(* CODESYS project tc3_bacnetrev14.library
   Company: Beckhoff Automation GmbH
   DefaultNamespace: Tc3_BACnetRev14
   Version: 4.0.11.0
   Placeholder: Tc3_BACnetRev14
   Author: Beckhoff Automation GmbH
   Description: The PLC library is a collection of function blocks for programming a BACnet controller. For each BACnet object function blocks are available that are read and written via the selected properties. In general a distinction is made between function blocks for server and client objects. Function blocks for client objects have the prefix "Remote", since they enable access to remote BACnet objects on other devices. The BACnet object function blocks ascertain whether process data are valid and the BACnet controller is ready for operation.
   Title: Tc3_BACnetRev14

Project tree, tasks and I/O mapping:
  libraries: Tc2_Standard, * (Beckhoff Automation GmbH); Tc2_System, * (Beckhoff Automation GmbH); Tc2_Utilities, * (Beckhoff Automation GmbH); Tc3_BA2_Common, * (Beckhoff Automation GmbH); Tc3_Module, * (Beckhoff Automation GmbH)
  DUTs/
    Enumerations/
      [Internal]/
        data type E_BACnet_CommMode
        data type E_BACnet_MultistateVal
        data type E_BACnet_PlcAction
      Properties/
        Calendar/
          data type E_BACnet_CalendarEntryChoice
          data type E_BACnet_CalendarEntryType
        DateTime/
          data type E_BACnet_DaysOfWeekBits
          data type E_BACnet_TimeStampChoice
        Error/
          data type E_BACnet_ErrorClass
          data type E_BACnet_ErrorCode
          data type E_BACnet_ErrorType
        Event/
          data type E_BACnet_EventState
          data type E_BACnet_EventTransitionBits
          data type E_BACnet_EventType
        LogBuffer/
          data type E_BACnet_LogRecordChoice
        Recipient/
          data type E_BACnet_AddressChoice
          data type E_BACnet_RecipientChoice
        Scheduler/
          data type E_BACnet_EnumerationValueChoice
          data type E_BACnet_SchedBType
          data type E_BACnet_SpecialEventChoice
          data type E_BACnet_ValueChoice
        data type E_BACnet_AbortReason
        data type E_BACnet_AdapterStatus
        data type E_BACnet_BinaryPV
        data type E_BACnet_DataTypes
        data type E_BACnet_DeviceStatus
        data type E_BACnet_FileAccessMethod
        data type E_BACnet_LifeSafetyMode
        data type E_BACnet_LifeSafetyOperation
        data type E_BACnet_LimitEnableBits
        data type E_BACnet_LoopMode
        data type E_BACnet_NodeType
        data type E_BACnet_NotifyType
        data type E_BACnet_ObjectSupportedBits
        data type E_BACnet_PersistentDataState
        data type E_BACnet_Priority
        data type E_BACnet_ProgramError
        data type E_BACnet_ProgramRequest
        data type E_BACnet_ProgramState
        data type E_BACnet_RejectReason
        data type E_BACnet_Reliability
        data type E_BACnet_Segmentation
        data type E_BACnet_ServicesSupportedBits
        data type E_BACnet_SilencedState
        data type E_BACnet_StatusFlags
        data type E_BACnet_StringEncodingTypes
      Remote/
        data type E_BACnetRM_ClientState
        data type E_BACnetRM_Error
        data type E_BACnetRM_RequestType
      data type E_BACnet_Error
    Interfaces/
      Remote/
        [Base]/
          interface I_BACnetRM_Object
        [Internal]/
          interface I_BACnetRM_BaseObject: OnCOV, OnReqError, Error, ObjectID, ObjectInstance, ObjectType, Ready
          interface I_BACnetRM_ObjectOwner: OnBACnetRMObjectCOV, OnBACnetRMObjectStateChanged, LogMsg
        interface I_BACnetRM_Req: Send, GetRequestType, IsReady
      Server/
        [Base]/
          interface I_BACnet_Object: Parent, Description, ObjectName
        [Internal]/
          interface I_BACnet_BaseObject: Error, ObjectID, ObjectInstance, ObjectType, Ready, ReadProperty, SyncPropertyCOV, WriteProperty
          interface I_BACnet_ObjectOwner: OnBACnetObjectStateChanged, LogMsg, SymbolPath
        Misc/
          interface I_BACnet_Cal
          interface I_BACnet_View
    Types/
      [ADS]/
        data type ST_BACnet_AdsConnection
        data type ST_BACnet_GlobalAdsBuffer
      [Internal]/
        ObjectList/
          data type ST_ObjectListEntry
      Diagnose/
        data type ST_BACnet_ConfirmedServiceDiag
        data type ST_BACnet_DiagEthStatistics
        data type ST_BACnet_Diagnosis
        data type ST_BACnet_DiagnosisTiming
        data type ST_BACnet_FrameStatistics
        data type ST_BACnet_Info
        data type ST_BACnet_ServerStatistics
        data type ST_BACnet_TcIoEthStatistic
        data type ST_BACnet_TcIoEthTxRxErrorCount
        data type ST_BACnet_UnConfirmedServiceDiag
      Properties/
        [ADS]/
          Calendar/
            data type ST_BACnet_CalendarEntry
            data type ST_BACnet_CalendarEntryDate
            data type ST_BACnet_CalendarEntryDateRange
            data type ST_BACnet_CalendarEntryWeekNDay
            data type T_BACnet_CalendarEntryTypeFilter
          DateTime/
            data type ST_BACnet_TimeStampDateTime
            data type ST_BACnet_TimeValue
            data type ST_BACnet_TimeValueBool
            data type ST_BACnet_TimeValueList
            data type ST_BACnet_TimeValueReal
          LogBuffer/
            data type ST_BACnet_LogBufferEntryReal
            data type ST_BACnet_LogBufferReal
          LogRecord/
            data type ST_BACnet_LogDatum
            data type ST_BACnet_LogDatumList
            data type ST_BACnet_LogRecord
            data type ST_BACnet_LogRecordList
          Schedule/
            data type ST_BACnet_DailySchedule
            data type ST_BACnet_ExceptionScheduleBool
            data type ST_BACnet_ExceptionScheduleCalDate
            data type ST_BACnet_ExceptionScheduleCalRef
            data type ST_BACnet_ExceptionScheduleCalWnD
            data type ST_BACnet_ExceptionScheduleEntryBool
            data type ST_BACnet_ExceptionScheduleEntryReal
            data type ST_BACnet_ExceptionScheduleReal
            data type ST_BACnet_Value
            data type ST_BACnet_ValueList
            data type ST_BACnet_WeeklyScheduleBool
            data type ST_BACnet_WeeklyScheduleReal
          ValidFields/
            data type ST_BACnet_ValidFields_DeviceObjectPropertyReference
          data type ST_BACnet_CharacterStringExt
          data type ST_BACnet_CharacterStringExtListEntry
          data type ST_BACnet_DeviceObjectPropertyReference
          data type ST_BACnet_DeviceObjectReference
          data type ST_BACnet_LimitEnable
          data type ST_BACnet_ObjectIdentifierList
        Calendar/
          data type T_BACnet_CalendarDateList
        Event/
          data type ST_BACnet_Event
          data type ST_BACnet_EventMessageTexts
          data type ST_BACnet_EventMessageTextStrings
          data type ST_BACnet_Events
          data type ST_BACnet_EventTimeStamps
        Recipient/
          data type ST_BACnet_Address
          data type ST_BACnet_Destination
          data type ST_BACnet_Recipient
          data type ST_BACnet_RecipientEntry
          data type ST_BACnet_ValidDays
        References/
          data type ST_BACnet_ObjectPropertyReference
        Scheduler/
          data type ST_BACnet_EnumerationValueType
          data type ST_BACnet_SchedCalendar
          data type ST_BACnet_SchedException
          data type ST_BACnet_SpecialEvent
          data type ST_BACnet_SpecialEventList
          data type T_BACnet_SchedCalendar
          data type T_BACnet_SchedExceptionEntryList
          data type T_BACnet_SchedExceptionList
          data type T_BACnet_SchedWeek
        TLog/
          data type T_BACnet_TLogBuffer
        data type ST_BACnet_EventTransitionBits
        data type ST_BACnet_ServicesSupportedBits
        data type T_BACnet_ObjectIdentifier
        data type T_BACnet_StateText
      Remote/
        [Internal]/
          data type ST_BACnetRM_CmdRealValue
          data type ST_BACnetRM_FifoEntry
          data type ST_BACnetRM_LastWriteValue
          data type ST_BACnetRM_PropertyValueList
          data type ST_BACnetRM_ReadEntry
          data type ST_BACnetRM_ReqPtr
          data type ST_BACnetRM_RpmListEntry
          data type ST_BACnetRM_ScanParameter
          data type ST_BACnetRM_WriteEntry
        data type ST_BACnetRM_ScanResult
  GVLs/
    global variables BACnet_Globals
    global variables BACnet_Param
  POUs/
    Helper/
      [internal]/
        Calendar/
          function F_BACnet_CopyDateListEntry [ST]
        Remote/
          function F_BACnetRM_IsErrorSet [ST]
        String/
          function F_BACnet_ChrStrExtLen [ST]
          function F_BACnet_DecodeUCS2 [ST]
          function F_BACnet_DecodeUCS4 [ST]
          function F_BACnet_DecodeUTF8 [ST]
          function F_BACnet_EncodeUTF8 [ST]
          function F_BACnet_GetUsedStateText [ST]
          function F_BACnet_GetUsedUDINT [ST]
          function F_BACnet_UCS2ToWin1252 [ST]
          function F_BACnet_Utf8ToWin1252 [ST]
          function F_BACnet_Win1252ToUCS2 [ST]
          function F_BACnet_Win1252ToUtf8 [ST]
        Validation-Functions/
          function F_BACnet_IsObjIdentifierValid [ST]
          function F_BACnet_IsPriorityValid [ST]
          function F_BACnet_IsSchedBTypeValid [ST]
        function F_BACnet_AlignedSize [ST]
        function F_BACnet_AnalogPV [ST]
        function F_BACnet_BitFieldBit [ST]
        function F_BACnet_ChangeBitFieldBit [ST]
        function F_BACnet_EndOf [ST]
        function F_BACnet_IsBitFieldBitSet [ST]
        function F_BACnet_IsBitFieldBitSetPtr [ST]
        function F_BACnet_NextListElem [ST]
        function F_BACnet_SetBitFieldBit [ST]
        function F_BACnet_SysTimeDiff [ST]
        function F_BACnet_UnSetBitFieldBit [ST]
      Flags/
        function F_BACnet_EventEnable [ST]
        function F_BACnet_EventTransitionFlags [ST]
        function F_BACnet_GetEventTransFlagsData [ST]
        function F_BACnet_GetLimitEnFlagsData [ST]
        function F_BACnet_GetStatusFlagsData [ST]
        function F_BACnet_LimitEnable [ST]
        function F_BACnet_LimitEnableFlags [ST]
        function F_BACnet_StatusFlags [ST]
      MultiState/
        function F_BACnet_EnMultiStatePV [ST]
        function F_BACnet_MultiStatePV [ST]
      NC/
        function F_BACnet_DeviceRecipient [ST]
        function F_BACnet_EthernetRecipient [ST]
        function F_BACnet_EthernetRecipientEx [ST]
      Real/
        function F_BACnet_EnRealPV [ST]
        function F_BACnet_IsFinite [ST]
        function F_BACnet_NAN [ST]
        function F_BACnet_RealEQ [ST]
        function F_BACnet_RealGE [ST]
        function F_BACnet_RealGT [ST]
        function F_BACnet_RealLE [ST]
        function F_BACnet_RealLT [ST]
        function F_BACnet_RealNothing [ST]
        function F_BACnet_RealNull [ST]
        function F_BACnet_RealPV [ST]
        function F_BACnet_RealToStr [ST]
      Scheduler/
        Calendar/
          function F_BACnet_SchedCalendar [ST]
        Exception/
          function F_BACnet_SchedEntry1xA [ST]
          function F_BACnet_SchedEntry1xB [ST]
          function F_BACnet_SchedEntry1xM [ST]
          function F_BACnet_SchedEntry3xA [ST]
          function F_BACnet_SchedEntry3xB [ST]
          function F_BACnet_SchedEntry3xM [ST]
          function F_BACnet_SchedEntry5xA [ST]
          function F_BACnet_SchedEntry5xB [ST]
          function F_BACnet_SchedEntry5xM [ST]
        Weekly/
          function F_BACnet_SchedWeekly1xA [ST]
          function F_BACnet_SchedWeekly1xB [ST]
          function F_BACnet_SchedWeekly1xM [ST]
          function F_BACnet_SchedWeekly3xA [ST]
          function F_BACnet_SchedWeekly3xB [ST]
          function F_BACnet_SchedWeekly3xM [ST]
          function F_BACnet_SchedWeekly5xA [ST]
          function F_BACnet_SchedWeekly5xB [ST]
          function F_BACnet_SchedWeekly5xM [ST]
      String/
        function F_BACnet_GetObjectIdString [ST]
        function block FB_BACnet_StringExtDecode [ST]
        function block FB_BACnet_StringExtEncode [ST]
      function F_BACnet_GetObjectListIndex [ST]
      function F_BACnet_GetObjId [ST]
      function F_BACnet_GetObjInstance [ST]
      function F_BACnet_GetObjType [ST]
      function block FB_BACnet_AccLimit [ST]
      function block FB_BACnet_AvgValue [ST]
      function block FB_BACnet_PidControl [ST]
      function block FB_BACnet_PT1 [ST]
    Local/
      Objects/
        [Base]/
          Basic/
            function block FB_BACnet_EventObject [ST]: OnObjectStateChanged, FB_init, AcknowledgePLC, AcknowledgeRm, IsReliable, AckedTransitions, EventState, StateFlags
            function block FB_BACnet_Object [ST]: OnBACnetObjectStateChanged, OnObjectStateChanged, ValidateReference, ConcatTitle, ValidateTitles, FB_init, LogMsg, Parent, SymbolPath, ReadPropertyExceptionSched, ReadPropertyReference, WritePropertyExceptionSched, WritePropertyReference, Description, ObjectName
          function block FB_BACnet_BaseAI [ST]: OnObjectStateChanged, FB_init
          function block FB_BACnet_BaseAO [ST]: OnObjectStateChanged, FB_init
          function block FB_BACnet_BaseBI [ST]: OnObjectStateChanged, FB_init
          function block FB_BACnet_BaseBO [ST]: OnObjectStateChanged, FB_init
          function block FB_BACnet_BaseMI [ST]: OnObjectStateChanged, FB_init, StateCount
          function block FB_BACnet_BaseMO [ST]: OnObjectStateChanged, FB_init, StateCount
          function block FB_BACnet_BaseSched [ST]: OnObjectStateChanged, FB_init, ReadContent, WriteContent
          function block FB_BACnet_BaseTLog [ST]: OnObjectStateChanged
        [Internal]/
          Property/
            Buffer/
              [Archiv]/
                function block FB_BACnet_WeeklyScheduleBuffer [ST]: FB_init, ResetValue
              Base/
                function block FB_BACnet_BaseArrayBuffer [ST]
                function block FB_BACnet_BaseListBuffer [ST]: ValidateInst
                function block FB_BACnet_BasePropertyBuffer [ST]: ReadValue, WriteValue, MemSet, MemSetBYTE, MemSetUDINT, MemSetUINT, MemSetULINT, ValidateInst, OnObjectStateChanged, ResetValue
              function block FB_BACnet_DateListBuffer [ST]: FB_init
              function block FB_BACnet_EventLogBuffer [ST]: ValidateInst, FB_init
              function block FB_BACnet_ExceptionScheduleBuffer [ST]: FB_init
              function block FB_BACnet_TLMBuffer [ST]: ValidateInst, FB_init, ResetValue
              function block FB_BACnet_TrendLogBuffer [ST]: ValidateInst, FB_init, ResetValue
          function block FB_BACnet_BaseObject [ST]: Close, Execute, View_RegisterChildObject, DeleteObject, Sched_ReadEntry, Sched_SetNextDay, Sched_SetNextTimeVal, Sched_WriteEntry, Trend_NextLogRecord, OnObjectStateChanged, OnPostOnlineChange, FB_exit, Acknowledge, Error, ObjectID, ObjectInstance, ObjectType, Ready, State, EnableProperty, SetPropertyCount, WriteProtectProperty, AddPropertyElement, AddPropertyElementPtr, RemoveArrayElements, RemoveListElements, SetNumberOfStates, ReadProperty, ReadPropertyAckedTransitions, ReadPropertyBool, ReadPropertyDateList, ReadPropertyEventEnable, ReadPropertyEventState, ReadPropertyEventTimeStamps, ReadPropertyExceptionSched, ReadPropertyLimitEnable, ReadPropertyLogBuffer, ReadPropertyNotifyType, ReadPropertyReal, ReadPropertyRecipientList, ReadPropertyReference, ReadPropertyStatusFlags, ReadPropertyString, ReadPropertyUDInt, ReadPropertyUnit, ReadPropertyWeeklySched, GetSyncHandleMode, AddListElement, ApplySyncHandler, EvaluatePropSync, RequestSyncHandlers, RequestSyncHandlersEx, SyncProperty, SyncPropertyCOV, SyncPropertyIdx, SyncPropertyList, SyncPropertyPvPrio, WriteProperty, WritePropertyBool, WritePropertyDateList, WritePropertyEventEnable, WritePropertyExceptionSched, WritePropertyLimitEnable, WritePropertyLogBuffer, WritePropertyNotifyType, WritePropertyNull, WritePropertyReal, WritePropertyRealPrio, WritePropertyRecipientList, WritePropertyReference, WritePropertyString, WritePropertyStringIdx, WritePropertyUDInt, WritePropertyUInt, WritePropertyUnit, WritePropertyValue, WritePropertyValueEx, WritePropertyWeeklySched
        5P/
          function block FB_BACnet_AO_IO5P [ST]: OnObjectStateChanged, ActivePrio, EnManualRm, ValManualRm
          function block FB_BACnet_AO_Raw5P [ST]: OnObjectStateChanged, ActivePrio, EnManualRm, ValManualRm
          function block FB_BACnet_AV_5P [ST]: OnObjectStateChanged, ActivePrio, EnManualRm, ValManualRm
          function block FB_BACnet_BO_IO5P [ST]: OnObjectStateChanged, ActivePrio, EnManualRm, ValManualRm
          function block FB_BACnet_BO_Raw5P [ST]: OnObjectStateChanged, ActivePrio, EnManualRm, ValManualRm
          function block FB_BACnet_BV_5P [ST]: OnObjectStateChanged, ActivePrio, EnManualRm, ValManualRm
          function block FB_BACnet_MO_IO5P [ST]: OnObjectStateChanged, ActivePrio, EnManualRm, ValManualRm
          function block FB_BACnet_MO_Raw5P [ST]: OnObjectStateChanged, ActivePrio, EnManualRm, ValManualRm
          function block FB_BACnet_MV_5P [ST]: OnObjectStateChanged, ActivePrio, EnManualRm, ValManualRm
        function block FB_BACnet_Acc [ST]: OnObjectStateChanged, FB_init
        function block FB_BACnet_AI [ST]: OnObjectStateChanged
        function block FB_BACnet_AI_IO [ST]: OnObjectStateChanged
        function block FB_BACnet_AI_Raw [ST]: OnObjectStateChanged
        function block FB_BACnet_AO_IO [ST]: OnObjectStateChanged
        function block FB_BACnet_AO_Raw [ST]: OnObjectStateChanged
        function block FB_BACnet_AV [ST]: OnObjectStateChanged, FB_init
        function block FB_BACnet_AV_Disp [ST]: OnObjectStateChanged, FB_init
        function block FB_BACnet_AV_Setp [ST]: OnObjectStateChanged, FB_init
        function block FB_BACnet_BI_IO [ST]: OnObjectStateChanged
        function block FB_BACnet_BI_Raw [ST]: OnObjectStateChanged
        function block FB_BACnet_BO_IO [ST]: OnObjectStateChanged
        function block FB_BACnet_BO_Raw [ST]: OnObjectStateChanged
        function block FB_BACnet_BV [ST]: OnObjectStateChanged, FB_init
        function block FB_BACnet_BV_Disp [ST]: OnObjectStateChanged, FB_init
        function block FB_BACnet_BV_Setp [ST]: OnObjectStateChanged, FB_init
        function block FB_BACnet_Cal [ST]: OnObjectStateChanged, FB_init, ReadContent, WriteContent
        function block FB_BACnet_Device [ST]: OnObjectStateChanged, FB_init, Location
        function block FB_BACnet_EventLog [ST]: OnObjectStateChanged, FB_init
        function block FB_BACnet_Loop [ST]: OnObjectStateChanged, FB_init, Mode, ProportionalBand
        function block FB_BACnet_MI_IO [ST]
        function block FB_BACnet_MI_Raw [ST]
        function block FB_BACnet_MO_IO [ST]: OnObjectStateChanged
        function block FB_BACnet_MO_Raw [ST]
        function block FB_BACnet_MV [ST]: OnObjectStateChanged, FB_init, StateCount
        function block FB_BACnet_MV_Disp [ST]: OnObjectStateChanged, FB_init, StateCount
        function block FB_BACnet_MV_Setp [ST]: OnObjectStateChanged, FB_init, StateCount
        function block FB_BACnet_NC [ST]: OnObjectStateChanged, FB_init
        function block FB_BACnet_PC [ST]: OnObjectStateChanged, FB_init
        function block FB_BACnet_Prog [ST]: OnObjectStateChanged, FB_init
        function block FB_BACnet_SchedA [ST]: OnObjectStateChanged, FB_init
        function block FB_BACnet_SchedB [ST]: OnObjectStateChanged, FB_init
        function block FB_BACnet_SchedM [ST]: OnObjectStateChanged, FB_init
        function block FB_BACnet_TLM [ST]: OnObjectStateChanged, FB_init
        function block FB_BACnet_TLog [ST]: OnObjectStateChanged, FB_init, DeviceObjectPropertyReference
        function block FB_BACnet_View [ST]: OnObjectStateChanged, FB_init
      function block FB_BACnet_Server [ST]: GetObject, RegisterObject, ObjectCount, ServerItf, BackupSTM, Reset, OnPostOnlineChange, FB_Exit, Error, IsValid, ReadPropertyUint
    Remote/
      Objects/
        Basic/
          [Base]/
            Basic/
              function block FB_BACnetRM_Object [ST]: OnBACnetRMObjectCOV, OnBACnetRMObjectStateChanged, FB_init, LogMsg
            function block FB_BACnetRM_BaseTLog [ST]: OnObjectStateChanged
            function block FB_BACnetRM_EventObject [ST]: OnObjectStateChanged, StateFlags
          [Internal]/
            function block FB_BACnetRM_BaseObject [ST]: OnCOV, OnReqError, OnObjectStateChanged, Error, ObjectID, ObjectInstance, ObjectType, Ready, SyncProperty, SyncPropertyPrio
          function block FB_BACnetRM_Acc [ST]: OnObjectStateChanged, FB_init
          function block FB_BACnetRM_AI [ST]: OnObjectStateChanged, FB_init
          function block FB_BACnetRM_AO [ST]: OnObjectStateChanged, FB_init
          function block FB_BACnetRM_AV [ST]: OnObjectStateChanged, FB_init
          function block FB_BACnetRM_AV_Disp [ST]: OnObjectStateChanged, FB_init
          function block FB_BACnetRM_AV_Setp [ST]: OnCOV, OnObjectStateChanged, FB_init
          function block FB_BACnetRM_BI [ST]: OnObjectStateChanged, FB_init
          function block FB_BACnetRM_BO [ST]: OnObjectStateChanged, FB_init
          function block FB_BACnetRM_BV [ST]: OnObjectStateChanged, FB_init
          function block FB_BACnetRM_BV_Disp [ST]: OnObjectStateChanged, FB_init
          function block FB_BACnetRM_BV_Setp [ST]: OnCOV, OnObjectStateChanged, FB_init
          function block FB_BACnetRM_Cal [ST]: OnObjectStateChanged, FB_init
          function block FB_BACnetRM_Device [ST]: OnObjectStateChanged, FB_init
          function block FB_BACnetRM_Loop [ST]: OnObjectStateChanged, FB_init
          function block FB_BACnetRM_MI [ST]: OnObjectStateChanged, FB_init
          function block FB_BACnetRM_MO [ST]: OnObjectStateChanged, FB_init
          function block FB_BACnetRM_MV [ST]: OnObjectStateChanged, FB_init
          function block FB_BACnetRM_MV_Disp [ST]: OnObjectStateChanged, FB_init
          function block FB_BACnetRM_MV_Setp [ST]: OnCOV, OnObjectStateChanged, FB_init
          function block FB_BACnetRM_NC [ST]: OnObjectStateChanged, FB_init
          function block FB_BACnetRM_PC [ST]: OnObjectStateChanged, FB_init
          function block FB_BACnetRM_Prog [ST]: OnObjectStateChanged, FB_init
          function block FB_BACnetRM_SchedA [ST]: OnObjectStateChanged, FB_init
          function block FB_BACnetRM_SchedB [ST]: OnObjectStateChanged, FB_init
          function block FB_BACnetRM_SchedM [ST]: OnObjectStateChanged, FB_init
          function block FB_BACnetRM_TLM [ST]: FB_init
          function block FB_BACnetRM_TLog [ST]: FB_init
        Convenience/
          function block FB_BACnetRM_CnvLoop [ST]: OnObjectStateChanged
      Requests/
        [Internal]/
          [Base]/
            function block FB_BACnetRM_BaseProperty [ST]: OnExecuteChange, Free, Busy, Error, IsValid, Ready, Request
            function block FB_BACnetRM_ReqBase [ST]: GetRequestType, IsReady, IsValid, Send
            function block FB_BACnetRM_ReqBasic [ST]: OnSendPropertyDataRequest, InitTimer, TcAddRef, TcQueryInterface, TcRelease, OnError, CopyRemoteData, ProcessResult, Send, StartTimer, GetRequestType, IsReady
          function block FB_BACnetRM_ReqAckAlarm [ST]: OnSendPropertyDataRequest, Send, TcAddRef, TcQueryInterface, TcRelease, UpdateTimeStamp, GetRequestType, IsReady
          function block FB_BACnetRM_ReqCov [ST]: AddCovSlave, Send, ProcessResult, StartTimer, FB_Exit, GetRequestType, IsReady, Master, SendSubscription
          function block FB_BACnetRM_ReqFifo [ST]: AddFifoReq, ProcessReadFifo, ProcessWriteFifo, FB_Exit, IsValid
          function block FB_BACnetRM_ReqListAdd [ST]: Send, ProcessResult, GetRequestType, IsReady
          function block FB_BACnetRM_ReqListRem [ST]: Send, ProcessResult, GetRequestType
          function block FB_BACnetRM_ReqRead [ST]: Send, OnError, ProcessResult, GetRequestType
          function block FB_BACnetRM_ReqRpm [ST]: Send, UpdateRequest, Free, OnError, ProcessResult, _WritePropEntry, FB_exit, GetRequestType
          function block FB_BACnetRM_ReqWpm [ST]: Send, UpdateRequest, Free, OnError, ProcessResult, FB_exit, GetRequestType
          function block FB_BACnetRM_ReqWrite [ST]: Send, OnError, ProcessResult, GetRequestType, IsReady
        function block FB_BACnetRM_ReadProperty [ST]: OnExecuteChange, Free, FB_exit, IsValid
        function block FB_BACnetRM_WriteProperty [ST]: OnExecuteChange, Free, FB_exit, IsValid
      function block FB_BACnet_Client [ST]: OnCOV, OnReqError, OnRequestComplete, AddFifoReadReq, AddFifoWriteReq, UpdateRequests, CreateReadReq, CreateReqList, DeleteReqList, OptimizeCOV, OnPostOnlineChange, FB_Exit, Error, ObjectID, ObjectInstance, ObjectType, OpenRequestCount, Ready, AddReadProp, AddWriteProp
    function block FB_BACnet_Adapter [ST]: FB_exit, FB_init, GetDiagnosis, ResetDiagnosis, Device, Error, GetScanResult, StartScan, StartScanEx, TimeSync
  TEST/
    TestPackage/
      Structure Samples/
        PRG02/
          TEMPLATES/
            Custom/
              H/
                HtgCirABC123/
                  function block FB_BA_HtgCirABC123 [CFC]: FB_init
                  function block FB_BA_HtgCirABC123_Vlv [CFC]: FB_init
                HtgCirTZU555/
                  function block FB_BA_HtgCirTZU555 [CFC]: FB_init
                  function block FB_BA_HtgCirTZU555_Pu [CFC]: FB_init
            Standard/
              AC/
                function block FB_BA_AC01 [CFC]: FB_init
              H/
                function block FB_BA_HtgCir01 [CFC]: FB_init
              Universal/
                Valve/
                  function block FB_Bnet_Vlv_014 [CFC]: FB_init
          program MAIN_PRG02 [ST]
      TEMPLATES/
        HeatSupply/
          HeatingCircuit/
            Plants/
              function block FB_Bnet_H_HtgCir_01 [CFC]: FB_init
            function block FB_Bnet_H_HtgCir_HtgLmt [CFC]: FB_init
            function block FB_Bnet_H_HtgCir_Sp [CFC]: FB_init
            function block FB_MMUX_R04 [ST]
            function block FB_Swi2P [ST]
          data type E_xEnergyLvl
          data type E_xEnergyLvlA
          function block FB_Bnet_H_OpM [CFC]: FB_init
          function block FB_PrioSwi_B04 [ST]
          function block FB_PrioSwi_UDI08 [ST]
        Internal/
          function block FB_BA_Server_NC01 [ST]
        Universal/
          AntiBlocking/
            function F_RemSecsTon [ST]
            function block FB_AntBlkg [ST]
            function block FB_Bnet_AntiBlocking [CFC]: FB_init
          Control/
            DelayOff/
              function block FB_Bnet_DlyOff [CFC]: FB_init
            Scale/
              function block FB_Bnet_Scale_04 [CFC]: FB_init
              function block FB_Chrct04 [ST]
          Pump/
            1st/
              function block FB_Bnet_Pu1st [CFC]: FB_init
          Valve/
            function block FB_Bnet_Vlv_013 [CFC]: FB_init
        global variables Const
      TestFBs/
        RT/
          function block FB_ArrayHtgCir [ST]: FB_init
          function block FB_ArrayTest [ST]: FB_init
        function block FB_ClientTest [ST]
      program _MAIN [ST]
      program CLIENT [ST]
      program PERFORMANCE [ST]
      program PERFORMANCE_MIX [ST]
      program PLANT_DEMO [ST]: FB_init
      program RT [ST]
    program CLIENT_Andreas [ST]
    program MAIN [ST]
  Version/
    global variables Global_Version
*)

// DUTs/Enumerations/[Internal]/E_BACnet_CommMode
{attribute 'hide'}
{attribute 'qualified_only'}
TYPE E_BACnet_CommMode :
(
	eAuto,
	eCov,
	eCovC,
	eCovU,
	eRp,
	eRpm
);
END_TYPE

// DUTs/Enumerations/[Internal]/E_BACnet_MultistateVal
{attribute 'hide'}
{attribute 'qualified_only'}
TYPE E_BACnet_MultistateVal:
(
	eNull					:= 16#0,
	eMin					:= 1,
	eNothing				:= 16#FFFFFFFF
) UDINT;
END_TYPE

// DUTs/Enumerations/[Internal]/E_BACnet_PlcAction
{attribute 'hide'}
{attribute 'qualified_only'}
TYPE E_BACnet_PlcAction :
(
	eIdle,
	eStart,
	eSuspend,
	eCreateFinish
) UINT;
END_TYPE

// DUTs/Enumerations/Properties/Calendar/E_BACnet_CalendarEntryChoice
{attribute 'qualified_only'}
TYPE E_BACnet_CalendarEntryChoice :
(
(*
	BACnetDate              DATE;
	BACnetDateRange   		dateRange;
	BACnetWeekNDay          weekNDay;
*)
	eDate,
	eDateRange,
	eWeekNDay
);
END_TYPE

// DUTs/Enumerations/Properties/Calendar/E_BACnet_CalendarEntryType
{attribute 'qualified_only'}
TYPE E_BACnet_CalendarEntryType : (* Not a BACnet-Stack type! *)
(
	eNone,
	eRef,
	eDate,
	eDateRange,
	eWeekNDay
);
END_TYPE

// DUTs/Enumerations/Properties/DateTime/E_BACnet_DaysOfWeekBits
{attribute 'qualified_only'}
TYPE E_BACnet_DaysOfWeekBits :
(
	Invalid		:= -1,
	
	eBitMonday		:= 0,
	eBitTuesday		:= 1,
	eBitWednesday	:= 2,
	eBitThursday	:= 3,
	eBitFriday		:= 4,
	eBitSaturday	:= 5,
	eBitSunday		:= 6
);
END_TYPE

// DUTs/Enumerations/Properties/DateTime/E_BACnet_TimeStampChoice
{attribute 'qualified_only'}
TYPE E_BACnet_TimeStampChoice :
(
	eTsTime,
    eSequenceNumber,
    eDateTime
);
END_TYPE

// DUTs/Enumerations/Properties/Error/E_BACnet_ErrorClass
{attribute 'qualified_only'}
TYPE E_BACnet_ErrorClass :
(
	eDevice					:= 0,
	eObject					:= 1,
	eProperty				:= 2,
	eResources				:= 3,
	eSecurity				:= 4,
	eServices				:= 5,
	eVt						:= 6,
	eCommunication			:= 7,
	
	eErrorClassUnknown	    := 255,
	eErrorClassNoError		:= 256 // own value
);
END_TYPE

// DUTs/Enumerations/Properties/Error/E_BACnet_ErrorCode
{attribute 'qualifiedOnly'}
TYPE E_BACnet_ErrorCode :
(
	eOther										:= 0,
	eAuthenticationFailed						:= 1,
	eConfigurationInProgress					:= 2,
	eDeviceBusy									:= 3,
	eDynamicCreationNotSupported				:= 4,
	eFileAccessDenied							:= 5,
	eIncompatibleSecurityLevels					:= 6,
	eInconsistentParameters						:= 7,
	eInconsistentSelectionCriterion				:= 8,
	eInvalidDataType							:= 9,
	eInvalidFileAccessMethod					:= 10,
	eInvalidFileStartPosition					:= 11,
	eInvalidOperatorName						:= 12,
	eInvalidParameterDataType					:= 13,
	eInvalidTimeStamp							:= 14,
	eKeyGenerationError							:= 15,
	eMissingRequiredParameter					:= 16,
	eNoObjectsOfSpecifiedType					:= 17,
	eNoSpaceForObject							:= 18,
	eNoSpaceToAddListElement					:= 19,
	eNoSpaceToWriteProperty						:= 20,
	eNoVTSessionsAvailable						:= 21,
	ePropertyIsNotAList							:= 22,
	eObjectDeletionNotPermitted					:= 23,
	eObjectIdentifierAlreadyExists				:= 24,
	eOperationalProblem							:= 25,
	ePasswordFailure							:= 26,
	eReadAccessDenied							:= 27,
	eSecurityNotSupported						:= 28,
	eServiceRequestDenied						:= 29,
	eTimeout									:= 30,
	eUnknownObject								:= 31,
	eUnknownProperty							:= 32,
	eUnknownVTClass								:= 34,
	eUnknownVTSession							:= 35,
	eUnsupportedObjectType						:= 36,
	eValueOutOfRange							:= 37,
	eVtSessionAlreadyClosed						:= 38,
	eVtSessionTerminationFailure				:= 39,
	eWriteAccessDenied							:= 40,
	eCharacterSetNotSupported					:= 41,
	eInvalidArrayIndex							:= 42,
	eCovSubscriptionFailed						:= 43,
	eNotCovProperty								:= 44,
	eOptionalFunctionalityNotSupported			:= 45,
	eInvalidConfigurationData					:= 46,
	eDatatypeNotSupported						:= 47,
	eDuplicateName								:= 48,
	eDuplicateObjectId							:= 49,
	ePropertyIsNotAnArray						:= 50,
	eAbortBufferOverflow						:= 51,
	eAbortInvalidAPDUInThisState				:= 52,
	eAbortPreemptedByHigherPriorityTask			:= 53,
	eAbortSegmentationNotSupported				:= 54,
	eAbortProprietary							:= 55,
	eAbortOther									:= 56,
	eInvalidTag									:= 57,
	eNetworkDown								:= 58,
	eRejectBufferOverflow						:= 59,
	eRejectInconsistentParameters				:= 60,
	eRejectInvalidParameterDataType				:= 61,
	eRejectInvalidTag							:= 62,
	eRejectMissingRequiredParameter				:= 63,
	eRejectParameterOutOfRange					:= 64,
	eRejectTooManyArguments						:= 65,
	eRejectUndefinedEnumeration					:= 66,
	eRejectUnrecognizedService					:= 67,
	eRejectProprietary							:= 68,
	eRejectOther								:= 69,
	eUnknownDevice								:= 70,
	eUnknownRoute								:= 71,
	eValueNotInitialized						:= 72,
	eInvalidEventState							:= 73,
	eNoAlarmConfigured							:= 74,
	eLogBufferFull								:= 75,
	eLoggedValuePurged							:= 76,
	eNoPropertySpecified						:= 77,
	eNotConfiguredForTriggeredLogging			:= 78,
	eUnknownSubscription						:= 79,
	eParameterOutOfRange						:= 80,
	eListElementNotFound						:= 81,
	eBusy										:= 82,
	eCommunicationDisabled						:= 83,
	eUnknownFileSize							:= 122,
	eAbortAPDUTooLong							:= 123,
	eAbortApplicationExceededReplyTime			:= 124,
	eAbortOutOfResources						:= 125,
	eAbortTsmTimeout							:= 126,
	eAbortWindowSizeOutOfRange					:= 127,
	eFileFull									:= 128,
	eInconsistentConfiguration					:= 129,
	eInconsistentObjectType						:= 130,
	eInternalError								:= 131,
	eNotConfigured								:= 132,
	eOutOfMemory 								:= 133,
	
	eErrorCodeNoError							:= 256  // own value
);
END_TYPE

// DUTs/Enumerations/Properties/Error/E_BACnet_ErrorType
{attribute 'qualified_only'}
TYPE E_BACnet_ErrorType :
(
	eTypeError,
	eTypeReject,
	eTypeAbort
);
END_TYPE

// DUTs/Enumerations/Properties/Event/E_BACnet_EventState
{attribute 'qualified_only'}
TYPE E_BACnet_EventState:
(
	eNormal := 0,
	eFault := 1,
	eOffnormal := 2,
	eHighLimit := 3,
	eLowLimit := 4,
	eLifeSafetyAlarm := 5
) UDINT;
END_TYPE

// DUTs/Enumerations/Properties/Event/E_BACnet_EventTransitionBits
{attribute 'qualified_only'}
TYPE E_BACnet_EventTransitionBits:
(
	Invalid			:= -1,
	
	eToOffnormal	:= 0,
	eToFault		:= 1,
	eToNormal		:= 2
);
END_TYPE

// DUTs/Enumerations/Properties/Event/E_BACnet_EventType
{attribute 'qualified_only'}
TYPE E_BACnet_EventType:
(
	Invalid := -1,
	
	eChangeOfBitstring := 0,
	eChangeOfState := 1,
	eChangeOfValue := 2,
	eCommandFailure := 3,
	eFloatingLimit := 4,
	eOutOfRange := 5,
	eComplexEventType := 6,
	eDeprecated7 := 7,
	eChangeOfLifeSafety := 8,
	eEnumeration := 9,
	eBufferReady := 10,
	eUnsignedRange := 11,
	eReserved12 := 12,
	eAccessEvent := 13,
	eDoubleOutOfRange := 14,
	eSignedOutOfRange := 15,
	eUnsignedOutOfRange := 16,
	eChangeOfCharacterstring := 17,
	eChangeOfStateFlags := 18
);
END_TYPE

// DUTs/Enumerations/Properties/LogBuffer/E_BACnet_LogRecordChoice
{attribute 'qualified_only'}
TYPE E_BACnet_LogRecordChoice :
(
(*
enum BACnetLogRecordChoice
{
      logStatus,              // [0] BACnetLogStatus,
      booleanValue,           // [1] BOOL,
      realValue,              // [2] REAL,
      enumValue,              // [3] ENUMERATED, __ Optionally limited to 32 bits
      unsignedValue,          // [4] Unsigned, __ Optionally limited to 32 bits
      signedValue,            // [5] INTEGER, __ Optionally limited to 32 bits
      bitstringValue,         // [6] BIT STRING, __ Optionally limited to 32 bits
      nullValue,              // [7] NULL,
      failure,                // [8] Error,
      timeChange,             // [9] REAL,
      anyValue,               // [10] ABSTRACT_SYNTAX.&Type __ Optional
};
*)
	eLogStatus 	:= 0, (* BACnetLogStatus *)
	eBooleanValue := 1, (*  BOOL, *)
	eRealValue	:= 2, (*  REAL, *)
	eEnumValue	:= 3, (*  ENUMERATED, __ Optionally limited TO 32 bits *)
	eUnsignedValue:= 4, (*  Unsigned, __ Optionally limited TO 32 bits *)
	eSignedValue	:= 5, (*  INTEGER, __ Optionally limited TO 32 bits *)
	eBitstringValue:= 6, (*  BIT STRING, __ Optionally limited TO 32 bits *)
	eNullValue	:= 7, (*  NULL, *)
	eFailure		:= 8, (*  Error, *)
	eTimeChange	:= 9, (*  REAL, *)
	eAnyValue		:= 10 (*  ABSTRACT_SYNTAX.&TYPE __ Optional *)
);
END_TYPE

// DUTs/Enumerations/Properties/Recipient/E_BACnet_AddressChoice
{attribute 'qualified_only'}
TYPE E_BACnet_AddressChoice :
(
	eEthernet:=0,
	eArcnet:=1,
	eMsTp:=2,
	eLonTalk:=3,
	eLonTalkNeuronId:=4,
	eAddress_3:=5,
	eAddress_4:=6,
	eAddress_5:=7,
	eBroadcast:=8
);
END_TYPE

// DUTs/Enumerations/Properties/Recipient/E_BACnet_RecipientChoice
{attribute 'qualified_only'}
TYPE E_BACnet_RecipientChoice :
(
	eDevice,
	eAddress
);
END_TYPE

// DUTs/Enumerations/Properties/Scheduler/E_BACnet_EnumerationValueChoice
{attribute 'qualified_only'}
TYPE E_BACnet_EnumerationValueChoice :
(
	  eEnum := 0,
      eBinaryPV := 1,
      eEngineeringUnits := 2
)UDINT;
END_TYPE

// DUTs/Enumerations/Properties/Scheduler/E_BACnet_SchedBType
{attribute 'qualified_only'}
{warning disable C0125}
TYPE E_BACnet_SchedBType :
(
	Invalid				:= 0,
	
	eBinaryPV			:= 1,
	eBool				:= 2,
	
	First				:= eBinaryPV,
	Last				:= eBool,
	Count				:= (Last - First + 1)
);
END_TYPE
{warning restore C0125}

// DUTs/Enumerations/Properties/Scheduler/E_BACnet_SpecialEventChoice
{attribute 'qualified_only'}
TYPE E_BACnet_SpecialEventChoice :
(
	eCalendarEntry,
	eCalendarReference
);
END_TYPE

// DUTs/Enumerations/Properties/Scheduler/E_BACnet_ValueChoice
{attribute 'qualified_only'}
{warning disable C0125}
TYPE E_BACnet_ValueChoice :
(
	Invalid						:= -1,
	
	eNullValue					:= 0,
	eBoolValue					:= 1,
	eUnsignedValue				:= 2,
	eSignedValue				:= 3,
	eRealValue					:= 4,
	eDoubleValue				:= 5,
	eOctedStringValue			:= 6,
	eCharStringValue			:= 7,
	eObjectIdentifierValue 		:= 8,		// but DataType is 0x0C
	eEnumerationValue			:= 9,
	eMaxBACnetValueChoice		:= 10
	
	//XFirst						:= eNullValue,
	//XLast						:= eMaxBACnetValueChoice,
	//Count						:= (Last - First + 1)
);
END_TYPE
{warning restore C0125}

// DUTs/Enumerations/Properties/E_BACnet_AbortReason
{attribute 'qualified_only'}
TYPE E_BACnet_AbortReason :
(
	eOther := 0,
	eBufferOverflow := 1,
	eInvalidAPDUInThisState := 2,
	ePreemptedByHigherPriorityTask := 3,
	eSegmentationNotSupported := 4,
	eWindowSizeOutOfRange := 7,
	eApplicationExceededReplyTime := 8,
	eOutOfResources := 9,
	eTSMTimeout := 10,
	eAPDUTooLong := 11,
	
	eNoError := 256
);
END_TYPE

// DUTs/Enumerations/Properties/E_BACnet_AdapterStatus
{attribute 'qualified_only'}
TYPE E_BACnet_AdapterStatus :
(
	eInit				:= 16#0,
	eCheckIpAddr		:= 16#1,
	eCheckParam			:= 16#2,
	eGetGatewayMAC		:= 16#3,
	eWaitGatewayMAC		:= 16#4,
	eComplete			:= 16#8
);
END_TYPE

// DUTs/Enumerations/Properties/E_BACnet_BinaryPV
{attribute 'qualified_only'}
TYPE E_BACnet_BinaryPV:
(
	eInactive := 0,
	eActive := 1,
	eNull := 2,
	eNothing := 16#FFFF
);
END_TYPE

// DUTs/Enumerations/Properties/E_BACnet_DataTypes
{attribute 'qualified_only'}
TYPE E_BACnet_DataTypes:
(
	Invalid := -1,
	
	eNull := 0,
	eBool := 1,
	eUnsignedInteger := 2,
	eSignedInteger := 3,
	eReal := 4,
	eDouble := 5,
	eOctetString := 6,
	eCharacterStringExt := 7,
	eBitString := 8,
	eEnumerated := 9,
	eDate := 10,
	eTime := 11,
	eObjectIdentifier := 12,
	eDateTime := 14,
	eArrayIndex := 15,
	eCalendarEntry := 16,
	eObjectType := 17,
	eEventTransitionBits := 18,
	eActionList := 19,
	eStatusFlags := 20,
	eEventState := 21,
	eReliability := 22,
	ePolarity := 23,
	eEngineeringUnits := 25,
	ePriorityValue := 26,
	eLimitEnable := 27,
	eNotifyType := 29,
	eTimeStamp := 30,
	eDeviceObjectPropertyReference := 31,
	eDeviceStatus := 32,
	eServicesSupported := 33,
	eObjectTypesSupported := 34,
	eSegmentation := 35,
	eVTClass := 36,
	eVTSession := 37,
	eSessionKey := 38,
	eRecipient := 39,
	eAddressBinding := 40,
	eCOVSubscription := 41,
	eEventType := 42,
	eEventParameter := 43,
	eFileAccessMethod := 44,
	eReadAccessSpecification := 45,
	eReadAccessResult := 46,
	eObjectPropertyReference := 47,
	eSetpointReference := 48,
	eDestination := 49,
	eProgramState := 50,
	eProgramRequest := 51,
	eProgramError := 52,
	eDateRange := 53,
	eDailySchedule := 54,
	eSpecialEvent := 55,
	eClientCOV := 56,
	eLogRecord := 57,
	eLifeSafetyState := 58,
	eLifeSafetyMode := 59,
	eSilencedState := 60,
	eLifeSafetyOperation := 61,
	eBinaryPV := 62,
	eDaysOfWeek := 63,
	eWeekNDay := 64,
	eTimeValue := 65,
	eValue := 66,
	eAddress := 67,
	ePropertyIdentifier := 68,
	eEnumerationValueType := 69,
	eBitFieldBit := 70,
	eLogDatum := 71,
	eAnyType := 72,
	ePresentValue := 73,
	eContextTag := 74,
	eValueChoice := 75,
	eLogStatus := 76,
	eRecipientProcess := 77,
	eSubscribeCOVPropertyRequest := 78,
	ePropertyReference := 79,
	ePropertyResult := 80,
	eDeviceObjectPropertyValue := 81,
	eCOVNotificationRequest := 82,
	eEventNotificationRequest := 83,
	eNotificationParameters := 84,
	eChangeOfBitstring := 85,
	eChangeOfState := 86,
	eChangeOfValue := 87,
	eCommandFailure := 88,
	eFloatingLimit := 89,
	eOutOfRange := 90,
	ePropertyValue := 91,
	eComplexTag := 92,
	eChangeOfLifeSafety := 93,
	eExtended := 94,
	eBufferReady := 95,
	eUnsignedRange := 96,
	ePropertyResultValue := 97,
	eServiceCOVPropSubscription := 98,
	eServiceCOVSubscription := 99,
	eCOVNotification := 100,
	eAcknowledgeAlarmRequest := 101,
	eVTOpenRequest := 102,
	ePrescale := 103,
	eScale := 104,
	eAction := 105,
	eError := 106,
	eErrorType := 107,
	eErrorClass := 108,
	eErrorCode := 109,
	eRejectReason := 110,
	eAbortReason := 111,
	eBDTEntry := 112,
	eIpEntry := 113,
	eMaskEntry := 114,
	eEthernetAddress := 115,
	eLonTalkAddress := 116,
	eLonTalkNeuronId := 117,
	eNodeType := 118,
	eDeviceObjectReference := 119,
	eActionCommand := 120,
	eGetEventInformation := 121,
	eGetEnrollmentSummaryCriteria := 122,
	eGetEnrollmentSummaryCriteriaResponse := 123,
	eDeviceCommunicationControl := 124,
	eInt16 := 125,
	eUInt16 := 126,
	eUInt8 := 127,
	eTypeInt8 := 128,
	eByte := 129,
	eFDTEntry := 130,
	eAddress_3 := 131,
	eAddress_4 := 132,
	eAddress_5 := 133,
	ePersistentDataState := 134,
	eFallbackRealValue := 135,
	eFallbackBinaryValue := 136,
	eRealNull := 137,						// PresentValue in AnalogObj
	eEnumeratedNull := 138,					// PresentValue in BinaryObj
	eUnsignedIntegerNull := 139,			// PresentValue in Multistate
	eUnknown := 140,
	eDiagnosisPerformance := 200,
	eDiagnosisEthStatistics := 201,
	eFrameStatistics := 202,
	eInfo := 203,
	eDiagnosis := 204,
	eTcIoEthStatistic := 205,
	eTcIoEthTxRxErrorCount := 206,
	eTcIoEthPortStatistic := 207,
	eServerStatistics := 208,
	eFrameServicesDiag := 209,
	eUnsignedIntegerArr := 258,
	eCharacterStringExtArr := 263,
	eObjectIdentifierArr := 268,
	eCalendarEntryArr := 272,
	eActionListArr := 275,
	ePriorityValueArr := 282,
	eTimeStampArr := 286,
	eDeviceObjectPropertyReferenceArr := 287,
	eVTClassArr := 292,
	eVTSessionArr := 293,
	eSessionKeyArr := 294,
	eRecipientArr := 295,
	eAddressBindingArr := 296,
	eCOVSubscriptionArr := 297,
	eReadAccessSpecificationArr := 301,
	eReadAccessResultArr := 302,
	eDestinationArr := 305,
	eSpecialEventArr := 311,
	eLogRecordArr := 313,
	eLifeSafetyStateArr := 314,
	eTimeValueArr := 321,
	eUnsignedIntegerList := 514,
	eCharacterStringExtList := 519,
	eReadAccessSpecificationList := 557,
	eReadAccessResultList := 558,
	eSpecialEventList := 567,
	eLogRecordList := 569,
	eTimeValueList := 577,
	eValueList := 578,
	eLogDatumList := 583,
	ePropertyReferenceList := 591,
	ePropertyResultList := 592,
	eCOVNotificationRequestList := 594,
	eEventNotificationRequestList := 595,
	ePropertyValueList := 603,
	eDailyScheduleList := 1089
);
END_TYPE

// DUTs/Enumerations/Properties/E_BACnet_DeviceStatus
{attribute 'qualified_only'}
TYPE E_BACnet_DeviceStatus:
(
	Invalid					:= -1,
	
	eOperational 			:= 0,
	eOperationalReadOnly	:= 1,
	eDownloadRequired 		:= 2,
	eDownloadInProgress 	:= 3,
	eNonOperational 		:= 4,
	eBackupInProgress 		:= 5
);
END_TYPE

// DUTs/Enumerations/Properties/E_BACnet_FileAccessMethod
{attribute 'qualified_only'}
TYPE E_BACnet_FileAccessMethod:
(
	Invalid := -1,
	
	eRecordAccess := 0,
	eStreamAccess := 1
);
END_TYPE

// DUTs/Enumerations/Properties/E_BACnet_LifeSafetyMode
{attribute 'qualified_only'}
TYPE E_BACnet_LifeSafetyMode:
(
	Invalid := -1,
	
	eOff := 0,
	eOn := 1,
	eTest := 2,
	eManned := 3,
	eUnmanned := 4,
	eArmed := 5,
	eDisarmed := 6,
	ePrearmed := 7,
	eSlow := 8,
	eFast := 9,
	eDisconnected := 10,
	eEnabled := 11,
	eModeDisabled := 12,
	eAutomaticReleaseDisabled := 13,
	eModeDefault := 14
);
END_TYPE

// DUTs/Enumerations/Properties/E_BACnet_LifeSafetyOperation
{attribute 'qualified_only'}
TYPE E_BACnet_LifeSafetyOperation:
(
	Invalid := -1,
	
	eNone := 0,
	eSilence := 1,
	eSilenceAnble := 2,
	eSilenceVisual := 3,
	eReset := 4,
	eResetAlarm := 5,
	eResetFault := 6,
	eUnsilence := 7,
	eUnsilenceAnble := 8,
	eUnsilenceVisual := 9
);
END_TYPE

// DUTs/Enumerations/Properties/E_BACnet_LimitEnableBits
{attribute 'qualified_only'}
TYPE E_BACnet_LimitEnableBits:
(
	Invalid := -1,
	
	eLowLimit := 0,
	eHighLimit := 1
);
END_TYPE

// DUTs/Enumerations/Properties/E_BACnet_LoopMode
{attribute 'qualified_only'}
TYPE E_BACnet_LoopMode :
(
	Invalid := -1,
	
	eNone,					// LOOP object has unknown parameter settings
	eIdeal,					// Controller is in ideal form: P, I and D are in parallel junktion; unit of P, I and D is [1] (Kp, Ki, Kd)
	eStandard				// Controller works in standard form (most industrial applications): P parameter is applied to I and D; unit of I and D is time based [s] (Kp, Ti, Td)
);
END_TYPE

// DUTs/Enumerations/Properties/E_BACnet_NodeType
{attribute 'qualified_only'}
TYPE E_BACnet_NodeType :
(
	Invalid := -1,
	
	eUnknown := 0,
	eSystem := 1,
	eNetwork := 2,
	eDevice := 3,
	eOrganizational := 4,
	eArea := 5,
	eEquipment := 6,
	ePoint := 7,
	eCollection := 8,
	eProperty := 9,
	eFunctional := 10,
	eOther := 11
);
END_TYPE

// DUTs/Enumerations/Properties/E_BACnet_NotifyType
{attribute 'qualified_only'}
TYPE E_BACnet_NotifyType:
(
	Invalid := -1,
	
	eAlarm := 0,
	eNotifyEvent := 1
	// ntAckNotification := 2
);
END_TYPE

// DUTs/Enumerations/Properties/E_BACnet_ObjectSupportedBits
{attribute 'qualified_only'}
TYPE E_BACnet_ObjectSupportedBits:
(
	eSuppInvalid := -1,
	
	eSuppAnalogInput := 0,
	eSuppAnalogOutput := 1,
	eSuppAnalogValue := 2,
	eSuppBinaryInput := 3,
	eSuppBinaryOutput := 4,
	eSuppBinaryValue := 5,
	eSuppCalendar := 6,
	eSuppCommand := 7,
	eSuppDevice := 8,
	eSuppEventEnrollment := 9,
	eSuppFile := 10,
	eSuppGroup := 11,
	eSuppLoop := 12,
	eSuppMultiStateInput := 13,
	eSuppMultiStateOutput := 14,
	eSuppNotificationClass := 15,
	eSuppProgr := 16,
	eSuppSchedule := 17,
	eSuppAveraging := 18,
	eSuppMultiStateValue := 19,
	eSuppTrendLog := 20,
	eSuppLifeSafetyPoint := 21,
	eSuppLifeSafetyZone := 22,
	eSuppAccumulator := 23,
	eSuppPulseConverter := 24,
	eSuppEventLog := 25,
	eSuppGlobalGroup := 26,
	eSuppTrendLogMultiple := 27,
	eSuppLoadControl := 28,
	eSuppStructuredView := 29,
	eSuppAccessDoor := 30,
	eSuppunassigend31 := 31,
	eSuppAccessCredential := 32,
	eSuppAccessPoint := 33,
	eSuppAccessRights := 34,
	eSuppAccessUser := 35,
	eSuppAccessZone := 36,
	eSuppCredentialDataInput := 37,
	eSuppNetworkSecurity := 38,
	eSuppBitStringValue := 39,
	eSuppCharacterStringValue := 40,
	eSuppDatePatternValue := 41,
	eSuppDateValue := 42,
	eSuppDateTimePatternValue := 43,
	eSuppDateTimeValue := 44,
	eSuppIntegerValue := 45,
	eSuppLargeAnalogValue := 46,
	eSuppOctetStringValue := 47,
	eSuppPositiveIntegerValue := 48,
	eSuppTimePatternValue := 49,
	eSuppTimeValue := 50,
	eSuppNetworkPort := 51,
	eSuppAlertEnrollment := 52,
	eSuppChannel := 53
);
END_TYPE

// DUTs/Enumerations/Properties/E_BACnet_PersistentDataState
{attribute 'qualified_only'}
TYPE E_BACnet_PersistentDataState :
(
	Invalid := -1,
	
	eDisabled,
	eInitialize,
	eNoChange,
	eReady,
	eWrite,
	eWriting
);
END_TYPE

// DUTs/Enumerations/Properties/E_BACnet_Priority
{attribute 'qualified_only'}
{warning disable C0125}
TYPE E_BACnet_Priority:
(
	Invalid			:= -1,
	
	eNone			:= 0,
	eP1				:= 1,
	eP2				:= 2,
	eP3				:= 3,
	eP4				:= 4,
	eP5				:= 5,
	eP6				:= 6,
	eP7				:= 7,
	eP8				:= 8,
	eP9				:= 9,
	eP10			:= 10,
	eP11			:= 11,
	eP12			:= 12,
	eP13			:= 13,
	eP14			:= 14,
	eP15			:= 15,
	eP16			:= 16,
	
	First			:= eP1,
	Last			:= eP16,
	Count			:= (Last - First + 1)
);
END_TYPE
{warning restore C0125}

// DUTs/Enumerations/Properties/E_BACnet_ProgramError
{attribute 'qualified_only'}
TYPE E_BACnet_ProgramError:
(
	Invalid := -1,
	
	eProgramNormal := 0,
	eLoadFailed := 1,
	eProgerrorInternal := 2,
	eProgram := 3,
	eOther := 4
);
END_TYPE

// DUTs/Enumerations/Properties/E_BACnet_ProgramRequest
{attribute 'qualified_only'}
TYPE E_BACnet_ProgramRequest:
(
	Invalid := -1,
	
	eReady := 0,
	eLoad := 1,
	eRun := 2,
	eHalt := 3,
	eRestart := 4,
	eUnload := 5
);
END_TYPE

// DUTs/Enumerations/Properties/E_BACnet_ProgramState
{attribute 'qualified_only'}
TYPE E_BACnet_ProgramState:
(
	Invalid := -1,
	
	eIdle := 0,
	eLoading := 1,
	eRunning := 2,
	eWaiting := 3,
	eHalted := 4,
	eUnloading := 5
);
END_TYPE

// DUTs/Enumerations/Properties/E_BACnet_RejectReason
{attribute 'qualified_only'}
TYPE E_BACnet_RejectReason :
(
	eOther := 0,
	eBufferOverflow := 1,
	eInconsistentParameters := 2,
	eInvalidParameterDataType := 3,
	eInvalidTag := 4,
	eMissingRequiredParameter := 5,
	eParameterOutOfRange := 6,
	eTooManyArguments := 7,
	eUndefinedEnumeration := 8,
	eUnrecognizedService := 9,
	//..
	
	eNoError := 256
);
END_TYPE

// DUTs/Enumerations/Properties/E_BACnet_Reliability
{attribute 'qualified_only'}
TYPE E_BACnet_Reliability:
(
	eNoFaultDetected := 0,
	eNoSensor := 1,
	eOverRange := 2,
	eUnderRange := 3,
	eOpenLoop := 4,
	eShortedLoop := 5,
	eNoOutput := 6,
	eUnreliableOther := 7,
	eProcessError := 8,
	eMultiStateFault := 9,
	eConfigurationError := 10,
	eReserved11 := 11,
	eCommunicationFailure := 12,
	eMemberFault := 13
);
END_TYPE

// DUTs/Enumerations/Properties/E_BACnet_Segmentation
{attribute 'qualified_only'}
TYPE E_BACnet_Segmentation:
(
	Invalid := -1,
	
	eBoth := 0,
	eTransmit := 1,
	eReceive := 2,
	eNo := 3
);
END_TYPE

// DUTs/Enumerations/Properties/E_BACnet_ServicesSupportedBits
{attribute 'qualified_only'}
TYPE E_BACnet_ServicesSupportedBits:
(
	eSuppInvalid := -1,
	
	eSuppAcknowledgeAlarm := 0,
	eSuppConfirmedCOVNotification := 1,
	eSuppConfirmedEventNotification := 2,
	eSuppGetAlarmSummary := 3,
	eSuppGetEnrollmentSummary := 4,
	eSuppSubscribeCOV := 5,
	eSuppAtomicReadFile := 6,
	eSuppAtomicWriteFile := 7,
	eSuppAddListElement := 8,
	eSuppRemoveListElement := 9,
	eSuppCreateObject := 10,
	eSuppDeleteObject := 11,
	eSuppReadProperty := 12,
	eSuppReadPropertyConditional := 13,
	eSuppReadPropertyMultiple := 14,
	eSuppWriteProperty := 15,
	eSuppWritePropertyMultiple := 16,
	eSuppDeviceCommunicationControl := 17,
	eSuppConfirmedPrivateTransfer := 18,
	eSuppConfirmedTextMessage := 19,
	eSuppReinitializeDevice := 20,
	eSuppVtOpen := 21,
	eSuppVtClose := 22,
	eSuppVtData := 23,
	eSuppAuthenticate := 24,
	eSuppRequestKey := 25,
	eSuppIAm := 26,
	eSuppIHave := 27,
	eSuppUnconfirmedCOVNotification := 28,
	eSuppUnconfirmedEventNotification := 29,
	eSuppUnconfirmedPrivateTransfer := 30,
	eSuppUnconfirmedTextMessage := 31,
	eSuppTimeSynchronization := 32,
	eSuppWhoHas := 33,
	eSuppWhoIs := 34,
	eSuppReadRange := 35,
	eSuppUtcTimeSynchronization := 36,
	eSuppLifeSafetyOperation := 37,
	eSuppSubscribeCOVProperty := 38,
	eSuppGetEventInformation := 39
);
END_TYPE

// DUTs/Enumerations/Properties/E_BACnet_SilencedState
{attribute 'qualified_only'}
TYPE E_BACnet_SilencedState:
(
	Invalid := -1,
	
	eUnsilenced := 0,
	eAnbleSilenced := 1,
	eVisibleSilenced := 2,
	eAllSilenced := 3
);
END_TYPE

// DUTs/Enumerations/Properties/E_BACnet_StatusFlags
{attribute 'qualified_only'}
TYPE E_BACnet_StatusFlags:
(
	Invalid := -1,
	
	eInAlarm := 0,
	eFault := 1,
	eOverridden := 2,
	eOutOfService := 3
);
END_TYPE

// DUTs/Enumerations/Properties/E_BACnet_StringEncodingTypes
{attribute 'qualified_only'}
TYPE E_BACnet_StringEncodingTypes :
(
	Invalid		:= -1,
	
	eAnsiUTF8	:= 0,
	eDBCS		:= 1,
	eJIS		:= 2,
	eUCS4		:= 3,
	eUCS2		:= 4,
	eISO8859	:= 5
);
END_TYPE

(*
---------------------------------------------
ISO8859
---------------------------------------------
						Part 1	Latin-1_ Western European__					
						Part 2	Latin-2_ Central European__					
						Part 3	Latin-3_ South European__					
						Part 4	Latin-4_ North European__					
Part 5	Latin/Cyrillic
Part 6	Latin/Arabic
Part 7	Latin/Greek
Part 8	Latin/Hebrew
						Part 9	Latin-5 _Turkish__					
						Part 10	Latin-6 _Nordic__					
Part 11	Latin/Thai
Part 12	"non-existent part" Latin/Devanagari
						Part 13	Latin-7_ Baltic Rim__					
						Part 14	Latin-8_ Celtic__					
Part 15	Latin-9
						Part 16	Latin-10_ South-Eastern European__					
---------------------------------------------
*)

// DUTs/Enumerations/Remote/E_BACnetRM_ClientState
{attribute 'qualified_only'}
TYPE E_BACnetRM_ClientState :
(
	eInit,
	eReadSupportedServices,
	eCalcAuto,
	eCreateRequests,
	eCycle,
	eReInit,
	eError
);
END_TYPE

// DUTs/Enumerations/Remote/E_BACnetRM_Error
{attribute 'qualified_only'}
TYPE E_BACnetRM_Error :
(
	eNone				:= 1,
	
	// General:
	eKillMe				:= 2,		// (BETA) ...
	eInvalidService 	:= 20
);
END_TYPE

// DUTs/Enumerations/Remote/E_BACnetRM_RequestType
{attribute 'qualified_only'}
TYPE E_BACnetRM_RequestType :
(
	eUndefined,
	
	eRead,
	eReadPropertyMultiple,
	eWrite,
	eWritePropertyMultiple,
	eCOV,
	eCOV_C,
	eCOV_U,
	eAcknowledge,
	eAddListElement,
	eRemoveListElement
);
END_TYPE

// DUTs/Enumerations/E_BACnet_Error
{attribute 'qualified_only'}
TYPE E_BACnet_Error :
(
	eNoError														:= 0,
	
	// General:
	eNoValidNetId													:= 1,
	eWrongMapping													:= 2,
	eOperational													:= 3,
	eNoEthLink														:= 4,
	eNoGateway														:= 5,
	eWocTriggerUnsup												:= 6,
	eWocDisabled													:= 7,
	eInvalidObjectId												:= 8,
	eInvalidObjectType												:= 10,
	eInvalidCycleTime												:= 11,
	eInvalidParameter												:= 12,
	eInvalidClient													:= 14,
	eInvalidServer													:= 15,
	eNotFoundBySymbol												:= 16,
	eCreateObject													:= 17,
	eDeviceNotFound													:= 18,

	// Errors with reset:
	ePersistentWrite												:= 20,
	eInvalidAdsConn													:= 21,
	eClientTimeout													:= 22,
	eClientService													:= 23,
	eWocTriggerActive												:= 24,
	eRevisionRead													:= 25,
	ePersistentPlcWrite												:= 26,
	eInvalidTask													:= 27,

	// ADS connection errors:
	eADS_NoValidNetId												:= 30,						// missing a valid Net ID
	eADS_Data														:= 31,						// ADS data length is wrong
	eADS_Read														:= 32,						// ADS read function was aborted
	eADS_Write														:= 33,						// ADS write function was aborted
	eADS_ObjType													:= 34,						// object type is wrong
	eADS_ObjListEmpty												:= 35,						// object list is empty
	eADS_DeviceOp													:= 36,						// device is not operational
	eADS_NoDevice													:= 37,						// no device object in object info list
	eADS_ObjInstance												:= 38,						// object list info is wrong
	eADS_AmsPort													:= 39,						// read AMS port is invalid (<1000)
	eADS_ObjectId													:= 40,						// object list info is wrong
	eADS_LegacyStack												:= 41,						// revision 6 stack detected (service is available from/above revision 9)
	eADS_ObjIdMissmatch												:= 42,						// object ID mapped and object list info are different
	eADS_BufferSize													:= 43,						// Property data larger than ADS buffer
	eADS_SchedData													:= 44,						// Wrong schedule property data
	eUnknownEventChoice												:= 45,						// Unknown event choice type
	eUnknownEntryChoice												:= 46,						// Unknown entry choice type
	eADS_TooManyObjects												:= 47,						// List of objects are longer than output list size
	eADS_WrongEntrySize												:= 48,						// expected entry size dosn't match read size
	eADS_RecipientData												:= 49,						// Invalid recipient data, device type expected
	eADS_TooManyEntries												:= 50,						// More entries than expected
	eADS_NotEnoughEntries											:= 51,						// Property incomplete, missing entries
	eADS_Encoding													:= 52,						// String encoding not supported
	eADS_NoServerClient												:= 53,						// Given ADS connection is not an server or client connection (expected bClient or bServer)
	eADS_NoNotificationSink											:= 54						// Given ADS connection is not an notification sink connection (expected bNSink)
);
END_TYPE

// DUTs/Types/[ADS]/ST_BACnet_AdsConnection
{attribute 'hide'}
TYPE ST_BACnet_AdsConnection :
STRUCT
	bValid		: BOOL; (* information are valid *)
	nReload		: USINT; (* reload counter *)
	sAmsNetId	: T_AmsNetId;
	nAmsPort	: T_AmsPort := 1000;
	bServer		: BOOL;
	bClient		: BOOL;
	bNSink		: BOOL;
	nDeviceId	: UDINT; (* Device object instance resp. BACnet ID *)
END_STRUCT
END_TYPE

// DUTs/Types/[ADS]/ST_BACnet_GlobalAdsBuffer
{attribute 'hide'}
TYPE ST_BACnet_GlobalAdsBuffer :
STRUCT
	bTestSet	: BOOL;
	nLocked		: DINT; (* -1 Buffer not ready, 0 Buffer ready, 1..n Buffer used (locked) *)
	arrData		: ARRAY[0..BACnet_Param.nADS_BufferSize] OF BYTE;
END_STRUCT
END_TYPE

// DUTs/Types/[Internal]/ObjectList/ST_ObjectListEntry
TYPE INTERNAL ST_ObjectListEntry :
STRUCT
	tObjectID : T_BACnet_ObjectIdentifier;
	pObject	  : I_BACnet_Object;
END_STRUCT
END_TYPE

// DUTs/Types/Diagnose/ST_BACnet_ConfirmedServiceDiag
{attribute 'hide'}
TYPE ST_BACnet_ConfirmedServiceDiag :
STRUCT
	nReqSend: DWORD; (* ULONG *)
	nReqSendFail: DWORD; (* ULONG *)
	nReqRecv: DWORD; (* ULONG *)
	nReqRecvFail: DWORD; (* ULONG *)
	nAckSend: DWORD; (* ULONG *)
	nAckSendFail: DWORD; (* ULONG *)
	nAckRecv: DWORD; (* ULONG *)
	nAckRecvFail: DWORD; (* ULONG *)
END_STRUCT
END_TYPE

// DUTs/Types/Diagnose/ST_BACnet_DiagEthStatistics
{attribute 'hide'}
TYPE ST_BACnet_DiagEthStatistics :
STRUCT
	ethStat: ST_BACnet_TcIoEthStatistic;
	txRxErrCnt: ST_BACnet_TcIoEthTxRxErrorCount;
END_STRUCT
END_TYPE

// DUTs/Types/Diagnose/ST_BACnet_Diagnosis
{attribute 'hide'}
TYPE ST_BACnet_Diagnosis :
STRUCT
	ethDevice: ST_BACnet_DiagEthStatistics;
	execTiming: ST_BACnet_DiagnosisTiming;
	frameStatistics: ST_BACnet_FrameStatistics;
	nRes1 : DWORD;
	info: ST_BACnet_Info;
	nRes2 : DWORD;
	serverInfo: ST_BACnet_ServerStatistics;
	lastUpdate: ST_BA_DateTime;
	nRes3 : DWORD;
END_STRUCT
END_TYPE

// DUTs/Types/Diagnose/ST_BACnet_DiagnosisTiming
{attribute 'hide'}
TYPE ST_BACnet_DiagnosisTiming :
STRUCT
	msIoInCurExecutionTime: DWORD; (* ULONG *)
	msIoInMinExecutionTime: DWORD; (* ULONG *)
	msIoInMaxExecutionTime: DWORD; (* ULONG *)
	msIoOutCurExecutionTime: DWORD; (* ULONG *)
	msIoOutMinExecutionTime: DWORD; (* ULONG *)
	msIoOutMaxExecutionTime: DWORD; (* ULONG *)
	msCycleCurExecutionTime: DWORD; (* ULONG *)
	msCycleMinExecutionTime: DWORD; (* ULONG *)
	msCycleMaxExecutionTime: DWORD; (* ULONG *)
	msInputCurDistanceTime: DWORD; (* ULONG *)
	msInputMinDistanceTime: DWORD; (* ULONG *)
	msInputMaxDistanceTime: DWORD; (* ULONG *)
END_STRUCT
END_TYPE

// DUTs/Types/Diagnose/ST_BACnet_FrameStatistics
{attribute 'hide'}
TYPE ST_BACnet_FrameStatistics :
STRUCT
	confirmed: ARRAY[0..29] OF ST_BACnet_ConfirmedServiceDiag; (* [SERVICE_CONFIRMED_MAX + 1]; 29 + 1 *)
	unConfirmed: ARRAY[0..9] OF ST_BACnet_UnConfirmedServiceDiag; (* [SERVICE_UNCONFIRMED_MAX + 1]; 9 *)
	nSegmSendTimeouts: DWORD; (* ULONG *)
	nFrameAllocFailCnt: DWORD; (* ULONG *)
	nFrameSendCnt: DWORD; (* ULONG *)
	nFrameSendFailCnt: DWORD; (* ULONG *)
	nFrameRecvCnt: DWORD; (* ULONG *)
	nFrameRecvFailCnt: DWORD; (* ULONG *)
	nLinkStatusChangedCnt: DWORD; (* ULONG *)
END_STRUCT
END_TYPE

// DUTs/Types/Diagnose/ST_BACnet_Info
{attribute 'hide'}
TYPE ST_BACnet_Info :
STRUCT
	nAmsAllocCnt: DINT; (* LONG *)
	nAmsAllocCntMax: DWORD; (* ULONG *)
	nAmsAllocFailCnt: DWORD; (* ULONG *)
	nAvailPhysMemBytes: DWORD; (* ULONG *)
	nAvailFlashMemBytes: ARRAY[0..1] OF DWORD; (* ULONGLONG *)
	nRecvFrameFifoSize: DWORD; (* ULONG *)
	nEmptyFrameFifoSize: DWORD; (* ULONG *)
	nRecvSegmUDPFramesListSize: DWORD; (* ULONG *)
	nRecvSegmFramesListSize: DWORD; (* ULONG *)
	nSendSegmFramesListSize: DWORD; (* ULONG *)
	nClientScanListSize: DWORD; (* ULONG *)
	nAmsRecvMissCount: DWORD; (* ULONG *)
END_STRUCT
END_TYPE

// DUTs/Types/Diagnose/ST_BACnet_ServerStatistics
{attribute 'hide'}
TYPE ST_BACnet_ServerStatistics :
STRUCT
	nOpenRequests: DWORD; (* ULONG *)
	nRequestRetries: DWORD; (* ULONG *)
	nRequestTimeOuts: DWORD; (* ULONG *)
	nPropChanges: DWORD; (* ULONG *)
	nPersistWrites: DWORD; (* ULONG *)
	persistChangeSetId: DWORD; (* ULONG *)
	secpersistNextWrite: DWORD; (* ULONG *)
	persistLastWrite: ST_BA_DateTime;
END_STRUCT
END_TYPE

// DUTs/Types/Diagnose/ST_BACnet_TcIoEthStatistic
{attribute 'hide'}
TYPE ST_BACnet_TcIoEthStatistic :
STRUCT
	dcTimeStamp: ARRAY[0..1] OF DWORD; (* ULONGLONG *)
	sendFrames: DWORD; (* ULONG *)
	recvFrames: DWORD; (* ULONG *)
	sendTimeRTime: DWORD; (* ULONG *)
	recvTimeRTime: DWORD; (* ULONG *)
	sendTimeNdis: DWORD; (* ULONG *)
	recvTimeNdis: DWORD; (* ULONG *)
END_STRUCT
END_TYPE

// DUTs/Types/Diagnose/ST_BACnet_TcIoEthTxRxErrorCount
{attribute 'hide'}
TYPE ST_BACnet_TcIoEthTxRxErrorCount :
STRUCT
	txCnt: DWORD; (* ULONG *)
	rxCnt: DWORD; (* ULONG *)
END_STRUCT
END_TYPE

// DUTs/Types/Diagnose/ST_BACnet_UnConfirmedServiceDiag
{attribute 'hide'}
TYPE ST_BACnet_UnConfirmedServiceDiag :
STRUCT
	nReqSend: DWORD; (* ULONG *)
	nReqSendFail: DWORD; (* ULONG *)
	nReqRecv: DWORD; (* ULONG *)
	nReqRecvFail: DWORD; (* ULONG *)
END_STRUCT
END_TYPE

// DUTs/Types/Properties/[ADS]/Calendar/ST_BACnet_CalendarEntry
TYPE ST_BACnet_CalendarEntry :
STRUCT
	eEventChoice		: E_BACnet_CalendarEntryChoice;
	{attribute 'hide'}
	_res1				: UINT;
	uCalEntry			: U_BA_DateVal;
END_STRUCT
END_TYPE

// DUTs/Types/Properties/[ADS]/Calendar/ST_BACnet_CalendarEntryDate
{attribute 'hide'}
TYPE ST_BACnet_CalendarEntryDate :
STRUCT
(*
	typedef struct _BACnetCalendarEntry
	{
	      BACnetCalendarEntryChoice choice;
	      union
	      {
	            BACnetDate              date;
	            BACnetDateRange   dateRange;
	            BACnetWeekNDay          weekNDay;
	      };
	}BACnetCalendarEntry, *PBACnetCalendarEntry;
*)
	eEntryChoice		: E_BACnet_CalendarEntryChoice;
	nRes				: WORD; (* ENUM alignment *)
	stDate				: ST_BA_Date;
END_STRUCT
END_TYPE

// DUTs/Types/Properties/[ADS]/Calendar/ST_BACnet_CalendarEntryDateRange
{attribute 'hide'}
TYPE ST_BACnet_CalendarEntryDateRange :
STRUCT
(*
	typedef struct _BACnetCalendarEntry
	{
	      BACnetCalendarEntryChoice choice;
	      union
	      {
	            BACnetDate              date;
	            BACnetDateRange   dateRange;
	            BACnetWeekNDay          weekNDay;
	      };
	}BACnetCalendarEntry, *PBACnetCalendarEntry;
*)
	eEntryChoice		: E_BACnet_CalendarEntryChoice;
	nRes				: WORD; (* ENUM alignment *)
	stStartDate			: ST_BA_Date;
	stEndDate			: ST_BA_Date;
END_STRUCT
END_TYPE

// DUTs/Types/Properties/[ADS]/Calendar/ST_BACnet_CalendarEntryWeekNDay
{attribute 'hide'}
TYPE ST_BACnet_CalendarEntryWeekNDay :
STRUCT
(*
	typedef struct _BACnetCalendarEntry
	{
	      BACnetCalendarEntryChoice choice;
	      union
	      {
	            BACnetDate              date;
	            BACnetDateRange   dateRange;
	            BACnetWeekNDay          weekNDay;
	      };
	}BACnetCalendarEntry, *PBACnetCalendarEntry;
*)
	eEntryChoice	: E_BACnet_CalendarEntryChoice;
	nRes1			: WORD; (* ENUM alignment *)
	nMonth			: USINT;
	nWeekOfMonth	: USINT;
	nDay			: USINT;
	nRes2			: USINT; (* weekNDay alignment *)
END_STRUCT
END_TYPE

// DUTs/Types/Properties/[ADS]/Calendar/T_BACnet_CalendarEntryTypeFilter
{attribute 'hide'}
TYPE T_BACnet_CalendarEntryTypeFilter : ARRAY[0..4] OF E_BACnet_CalendarEntryType; END_TYPE

// DUTs/Types/Properties/[ADS]/DateTime/ST_BACnet_TimeStampDateTime
{attribute 'hide'}
TYPE ST_BACnet_TimeStampDateTime :
STRUCT
	eType		: E_BACnet_TimeStampChoice;
	_fillBytes	: WORD;
	stDateTime	: ST_BA_DateTime;
END_STRUCT
END_TYPE

// DUTs/Types/Properties/[ADS]/DateTime/ST_BACnet_TimeValue
{attribute 'hide'}
TYPE ST_BACnet_TimeValue :
STRUCT
	stTime	: ST_BA_Time;
	nRes	: DWORD;
	stValue	: ST_BACnet_Value;
END_STRUCT
END_TYPE

// DUTs/Types/Properties/[ADS]/DateTime/ST_BACnet_TimeValueBool
{attribute 'hide'}
TYPE ST_BACnet_TimeValueBool :
STRUCT
	bValid		: BOOL;
	stTime		: ST_BA_Time;
	eType		: E_BACnet_DataTypes;
	bValue		: BOOL;
END_STRUCT
END_TYPE

// DUTs/Types/Properties/[ADS]/DateTime/ST_BACnet_TimeValueList
{attribute 'hide'}
TYPE ST_BACnet_TimeValueList :
STRUCT
	nEntrySize	: DWORD;
	nRes		: DWORD;
	stListEntry	: ST_BACnet_TimeValue;
END_STRUCT
END_TYPE

// DUTs/Types/Properties/[ADS]/DateTime/ST_BACnet_TimeValueReal
{attribute 'hide'}
TYPE ST_BACnet_TimeValueReal :
STRUCT
	bValid		: BOOL;
	stTime		: ST_BA_Time;
	eType		: E_BACnet_DataTypes;
	fValue		: REAL;
END_STRUCT
END_TYPE

// DUTs/Types/Properties/[ADS]/LogBuffer/ST_BACnet_LogBufferEntryReal
{attribute 'hide'}
TYPE ST_BACnet_LogBufferEntryReal :
STRUCT
	nTimeStamp	: DWORD; (* 100ms since 1900 *)
	stDateTime	: ST_BA_DateTime; (* BACnet time stamp *)
	fValue		: REAL;
END_STRUCT
END_TYPE

// DUTs/Types/Properties/[ADS]/LogBuffer/ST_BACnet_LogBufferReal
{attribute 'hide'}
TYPE ST_BACnet_LogBufferReal :
STRUCT
	nGet		: USINT; (* Update date counter *)
	sObjectDesc	: T_MAXSTRING; (* Object description *)
	nCount		: UDINT; (* log buffer entries *)
	arrEntries	: ARRAY[0..BACnet_Globals.nDataField_MaxLogBufferEntries] OF ST_BACnet_LogBufferEntryReal;
END_STRUCT
END_TYPE

// DUTs/Types/Properties/[ADS]/LogRecord/ST_BACnet_LogDatum
{attribute 'hide'}
TYPE ST_BACnet_LogDatum :
STRUCT
(*

typedef struct _BACnetLogDatum
{
      BACnetLogRecordChoice choice;
      union
      {
            DWORD logStatus; // BitString ... of type BACnetLogStatus
            BOOL booleanValue;
            FLOAT realValue;
            EnumerationValueType enumerationValue;
            ULONG unsignedValue;
            DWORD signedValue;
            DWORD bitstringValue;
            DWORD nullValue;
            BACnetError failure; 
            FLOAT timeChange;
            AnyType anyValue; // ABSTRACT-SYNTAX.&Type
      };
}BACnetLogDatum, *PBACnetLogDatum;

*)
	choice	: E_BACnet_LogRecordChoice;
	nRes	: WORD; (* ENUM alignment to 4 byte *)
	nData	: ARRAY[0..4] OF DWORD; (* 20 byte min. size - data type depending on choice selection *)
END_STRUCT
END_TYPE

// DUTs/Types/Properties/[ADS]/LogRecord/ST_BACnet_LogDatumList
{attribute 'hide'}
TYPE ST_BACnet_LogDatumList :
STRUCT
(*

typedef struct _BACnetLogDatumList
{
      DWORD nEntrySize; // 0x80000000 -> next entry
      DWORD reserved;
      BACnetLogDatum listEntry;
}BACnetLogDatumList, *PBACnetLogDatumList;

*)
	nEntrySize	: DWORD; (* 0x80000000 -> next entry *)
	reserved	: DWORD;
	listEntry	: ST_BACnet_LogDatum; (* first entry of log datum list *)
END_STRUCT
END_TYPE

// DUTs/Types/Properties/[ADS]/LogRecord/ST_BACnet_LogRecord
{attribute 'hide'}
TYPE ST_BACnet_LogRecord :
STRUCT
(*

typedef STRUCT _BACnetLogRecord
{
      ULONG validFields;
      BACnetDateTime timestamp;          // [0]
      DWORD statusFlags;                       // [2] optional
      BACnetLogDatumList logDatum;  // [1]
}BACnetLogRecord, *PBACnetLogRecord;

*)
	validFields	: UDINT;
	timestamp	: ST_BA_DateTime;
	statusFlags	: DWORD;
	logDatum	: ST_BACnet_LogDatumList;
END_STRUCT
END_TYPE

// DUTs/Types/Properties/[ADS]/LogRecord/ST_BACnet_LogRecordList
{attribute 'hide'}
TYPE ST_BACnet_LogRecordList :
STRUCT
(*

typedef struct _BACnetLogRecordList
{
      DWORD nEntrySize; // 0x80000000 -> next entry
      DWORD nSequence;  // "reserved"     -> Number of Sequence begins with 1
      BACnetLogRecord listEntry;
}BACnetLogRecordList, *PBACnetLogRecordList;

*)
	nEntrySize	: DWORD; (* 16#80000000 -> next entry *)
	nSequence	: DWORD; (* "reserved"  -> Number OF Sequence begins with 1 *)
	listEntry	: ST_BACnet_LogRecord; (* first entry of record list *)
END_STRUCT
END_TYPE

// DUTs/Types/Properties/[ADS]/Schedule/ST_BACnet_DailySchedule
{attribute 'hide'}
TYPE ST_BACnet_DailySchedule :
STRUCT
(*
	PropWeeklySchedule:
	
	typedef struct _BACnetDailySchedule
	{
	      DWORD nEntrySize; // 0x80000000 -> next entry
	      DWORD reserved;
	      BACnetTimeValueList listEntry;
	} BACnetDailySchedule, *PBACnetDailySchedule;
*)
	nEntrySize	: DWORD;
	nRes		: DWORD;
	stListEntry	: ST_BACnet_TimeValueList;
END_STRUCT
END_TYPE

// DUTs/Types/Properties/[ADS]/Schedule/ST_BACnet_ExceptionScheduleBool
{attribute 'hide'}
TYPE ST_BACnet_ExceptionScheduleBool :
STRUCT
	bReqGet		: BOOL; (* set TRUE if property should reloaded, TRUE --> FALSE = request accepted (starting reload) *)
	bReqSet		: BOOL; (* set TRUE for property write request, TRUE --> FALSE = request accepted (starting storage) *)
	nGet		: USINT; (* reload counter, count up if property was loaded successful *)
	nSet		: USINT; (* save counter, count up if property was stored successful *)
	bBusy		: BOOL; (* started writing data into "arrEntries", don't write data to avoid concurrent access *)
	arrEntries	: ARRAY[0..BACnet_Globals.nDataField_MaxExSchEntries] OF ST_BACnet_ExceptionScheduleEntryBool;
END_STRUCT
END_TYPE

// DUTs/Types/Properties/[ADS]/Schedule/ST_BACnet_ExceptionScheduleCalDate
{attribute 'hide'}
TYPE ST_BACnet_ExceptionScheduleCalDate :
STRUCT
	stStart			: ST_BA_Date;
	stEnd			: ST_BA_Date;
END_STRUCT
END_TYPE

// DUTs/Types/Properties/[ADS]/Schedule/ST_BACnet_ExceptionScheduleCalRef
{attribute 'hide'}
TYPE ST_BACnet_ExceptionScheduleCalRef :
STRUCT
	tCalObjectId	: T_BACnet_ObjectIdentifier := 16#FFFFFFFF;
END_STRUCT
END_TYPE

// DUTs/Types/Properties/[ADS]/Schedule/ST_BACnet_ExceptionScheduleCalWnD
{attribute 'hide'}
TYPE ST_BACnet_ExceptionScheduleCalWnD :
STRUCT
	nMonth			: USINT; (* 255 = all months of year *)
	nWeekOfMonth	: USINT; (* 255 = all weeks of month *)
	nDay			: USINT; (* 255 = all days of month *)
END_STRUCT
END_TYPE

// DUTs/Types/Properties/[ADS]/Schedule/ST_BACnet_ExceptionScheduleEntryBool
{attribute 'hide'}
TYPE ST_BACnet_ExceptionScheduleEntryBool :
STRUCT
	eEntryType		: E_BACnet_CalendarEntryType;
	ePriority		: E_BACnet_Priority;
	stDate			: ST_BACnet_ExceptionScheduleCalDate; (* date / date range *)
	stWeekNDay		: ST_BACnet_ExceptionScheduleCalWnD; (* week and day *)
	stCalRef		: ST_BACnet_ExceptionScheduleCalRef; (* week and day *)
	arrTimeValue	: ARRAY[0..BACnet_Globals.nDataField_MaxTimeValues] OF ST_BACnet_TimeValueBool;
END_STRUCT
END_TYPE

// DUTs/Types/Properties/[ADS]/Schedule/ST_BACnet_ExceptionScheduleEntryReal
{attribute 'hide'}
TYPE ST_BACnet_ExceptionScheduleEntryReal :
STRUCT
	eEntryType		: E_BACnet_CalendarEntryType;
	ePriority		: E_BACnet_Priority;
	stDate			: ST_BACnet_ExceptionScheduleCalDate; (* date / date range *)
	stWeekNDay		: ST_BACnet_ExceptionScheduleCalWnD; (* week and day *)
	stCalRef		: ST_BACnet_ExceptionScheduleCalRef; (* week and day *)
	arrTimeValue	: ARRAY[0..BACnet_Globals.nDataField_MaxTimeValues] OF ST_BACnet_TimeValueReal;
END_STRUCT
END_TYPE

// DUTs/Types/Properties/[ADS]/Schedule/ST_BACnet_ExceptionScheduleReal
{attribute 'hide'}
TYPE ST_BACnet_ExceptionScheduleReal :
STRUCT
	bReqGet		: BOOL; (* set TRUE if property should reloaded, TRUE --> FALSE = request accepted (starting reload) *)
	bReqSet		: BOOL; (* set TRUE for property write request, TRUE --> FALSE = request accepted (starting storage) *)
	nGet		: USINT; (* reload counter, count up if property was loaded successful *)
	nSet		: USINT; (* save counter, count up if property was stored successful *)
	bBusy		: BOOL; (* started writing data into "arrEntries", don't write data to avoid concurrent access *)
	arrEntries	: ARRAY[0..BACnet_Globals.nDataField_MaxExSchEntries] OF ST_BACnet_ExceptionScheduleEntryReal;
END_STRUCT
END_TYPE

// DUTs/Types/Properties/[ADS]/Schedule/ST_BACnet_Value
{attribute 'hide'}
TYPE ST_BACnet_Value :
STRUCT
	eValueChoice	: E_BACnet_ValueChoice;
	nRes1			: WORD; (* ENUM alignment *)
	nSize			: DWORD;
	stValue			: ST_BACnet_EnumerationValueType;
END_STRUCT
END_TYPE

// DUTs/Types/Properties/[ADS]/Schedule/ST_BACnet_ValueList
{attribute 'hide'}
TYPE ST_BACnet_ValueList :
STRUCT
	nEntrySize	: DWORD; (* 0x80000000 -> next entry *)
	reserved	: DWORD;
	listEntry	: ST_BACnet_Value; (* first entry of value list *)
END_STRUCT
END_TYPE

// DUTs/Types/Properties/[ADS]/Schedule/ST_BACnet_WeeklyScheduleBool
{attribute 'hide'}
TYPE ST_BACnet_WeeklyScheduleBool :
STRUCT
	bReqGet		: BOOL; (* set TRUE if property should reloaded, TRUE --> FALSE = request accepted (reload started) *)
	bReqSet		: BOOL; (* set TRUE for property write request, TRUE --> FALSE = request accepted (storage started) *)
	nGet		: USINT; (* reload counter, count up if property was loaded successful *)
	nSet		: USINT; (* save counter, count up if property was stored successful *)
	bBusy		: BOOL; (* started writing/reading data into/from "arrEntries", don't change data to avoid concurrent access *)
	arrEntries	: ARRAY[0..6] OF ARRAY[0..BACnet_Globals.nDataField_MaxDayEntry] OF ST_BACnet_TimeValueBool;
END_STRUCT
END_TYPE

// DUTs/Types/Properties/[ADS]/Schedule/ST_BACnet_WeeklyScheduleReal
{attribute 'hide'}
TYPE ST_BACnet_WeeklyScheduleReal :
STRUCT
	bReqGet		: BOOL; (* set TRUE if property should reloaded, TRUE --> FALSE = request accepted (reload started) *)
	bReqSet		: BOOL; (* set TRUE for property write request, TRUE --> FALSE = request accepted (storage started) *)
	nGet		: USINT; (* reload counter, count up if property was loaded successful *)
	nSet		: USINT; (* save counter, count up if property was stored successful *)
	bBusy		: BOOL; (* started writing/reading data into/from "arrEntries", don't change data to avoid concurrent access *)
	arrEntries	: ARRAY[0..6] OF ARRAY[0..BACnet_Globals.nDataField_MaxDayEntry] OF ST_BACnet_TimeValueReal;
END_STRUCT
END_TYPE

// DUTs/Types/Properties/[ADS]/ValidFields/ST_BACnet_ValidFields_DeviceObjectPropertyReference
{attribute 'hide'}
TYPE ST_BACnet_ValidFields_DeviceObjectPropertyReference :
STRUCT
	bObjectId				: BIT;
	bPropertyIdentifier		: BIT;

	{attribute 'hide'}
	nReserve1				: BIT;
	{attribute 'hide'}
	nReserve2				: BIT;
	{attribute 'hide'}
	nReserve3				: BIT;
	{attribute 'hide'}
	nReserve4				: BIT;
	{attribute 'hide'}
	nReserve5				: BIT;
	{attribute 'hide'}
	nReserve6				: BIT;
END_STRUCT
END_TYPE

// DUTs/Types/Properties/[ADS]/ST_BACnet_CharacterStringExt
{attribute 'hide'}
TYPE ST_BACnet_CharacterStringExt :
STRUCT
	cookie		: BYTE; (* 0 -> DO differentiate normal strings *)
	encoding	: BYTE;
	strLen		: UINT;
	stringData	: ARRAY[1..BACnet_Globals.nBACnetString_MaxLength] OF BYTE;
END_STRUCT
END_TYPE

// DUTs/Types/Properties/[ADS]/ST_BACnet_CharacterStringExtListEntry
{attribute 'hide'}
TYPE ST_BACnet_CharacterStringExtListEntry :
STRUCT
(* list header *)
	nEntrySize	: DWORD; (* byte size of data *)
	hdrInfo		: DWORD;
(* data *)
	extString	: ST_BACnet_CharacterStringExt;
END_STRUCT
END_TYPE

// DUTs/Types/Properties/[ADS]/ST_BACnet_DeviceObjectPropertyReference
{attribute 'hide'}
TYPE ST_BACnet_DeviceObjectPropertyReference :
STRUCT
	stValidFields			: ST_BACnet_ValidFields_DeviceObjectPropertyReference;
	tObjId					: T_BACnet_ObjectIdentifier;
	ePropIdentifier			: E_BACnetPropIdentifier;
	{attribute 'hide'}
	nReserve				: UINT;
	dwPropertyArrayIndex	: DWORD;
	tDeviceId				: T_BACnet_ObjectIdentifier;
END_STRUCT
END_TYPE

// DUTs/Types/Properties/[ADS]/ST_BACnet_DeviceObjectReference
{attribute 'hide'}
TYPE ST_BACnet_DeviceObjectReference :
STRUCT
	validFields : UDINT := 2;
	deviceId : T_BACnet_ObjectIdentifier;
	objId : T_BACnet_ObjectIdentifier;
END_STRUCT
END_TYPE

// DUTs/Types/Properties/[ADS]/ST_BACnet_LimitEnable
{attribute 'hide'}
TYPE ST_BACnet_LimitEnable:
STRUCT
	lowLimitEnable : BOOL;
	highLimitEnable : BOOL;
END_STRUCT
END_TYPE

// DUTs/Types/Properties/[ADS]/ST_BACnet_ObjectIdentifierList
{attribute 'hide'}
TYPE ST_BACnet_ObjectIdentifierList :
STRUCT
	nEntries	: UDINT;
	arrObjList	: ARRAY[0..BACnet_Globals.nDataField_MaxObjIdList] OF T_BACnet_ObjectIdentifier :=[ 16#FFFFFFFF];
END_STRUCT
END_TYPE

// DUTs/Types/Properties/Calendar/T_BACnet_CalendarDateList
TYPE T_BACnet_CalendarDateList : ARRAY[1 .. BACnet_Param.nCal_DateListCount] OF ST_BA_CalendarEntry; END_TYPE

// DUTs/Types/Properties/Event/ST_BACnet_Event
TYPE ST_BACnet_Event :
STRUCT
	acked : BOOL;
	message : STRING;
	timeStamp : DT;
	{attribute 'hide'} 
    {attribute 'tc_no_symbol'}
	bacnetTime : ST_BACnet_TimeStampDateTime;
END_STRUCT
END_TYPE

// DUTs/Types/Properties/Event/ST_BACnet_EventMessageTexts
TYPE ST_BACnet_EventMessageTexts :
STRUCT
	toOffNormal : ST_BACnet_CharacterStringExtListEntry;
	toFault : ST_BACnet_CharacterStringExtListEntry;
	toNormal : ST_BACnet_CharacterStringExtListEntry;
END_STRUCT
END_TYPE

// DUTs/Types/Properties/Event/ST_BACnet_EventMessageTextStrings
TYPE ST_BACnet_EventMessageTextStrings :
STRUCT
	toOffNormal : STRING;
	toFault : STRING;
	toNormal : STRING;
END_STRUCT
END_TYPE

// DUTs/Types/Properties/Event/ST_BACnet_Events
TYPE ST_BACnet_Events :
STRUCT
	toOffNormal : ST_BACnet_Event;
	toFault : ST_BACnet_Event;
	toNormal : ST_BACnet_Event;
END_STRUCT
END_TYPE

// DUTs/Types/Properties/Event/ST_BACnet_EventTimeStamps
TYPE ST_BACnet_EventTimeStamps :
STRUCT
	toOffNormal : ST_BACnet_TimeStampDateTime;
	toFault : ST_BACnet_TimeStampDateTime;
	toNormal : ST_BACnet_TimeStampDateTime;
END_STRUCT
END_TYPE

// DUTs/Types/Properties/Recipient/ST_BACnet_Address
{attribute 'hide'}
TYPE ST_BACnet_Address :
STRUCT
	eChoice : E_BACnet_AddressChoice;
	{attribute 'hide'}
	res0 : UINT;
	eAddress : ARRAY [0..7] OF BYTE;
	nNetworkNr : UINT;
END_STRUCT
END_TYPE

// DUTs/Types/Properties/Recipient/ST_BACnet_Destination
{attribute 'hide'}
TYPE ST_BACnet_Destination :
STRUCT
	stValidDays			: ST_BACnet_ValidDays;
	{attribute 'hide'}
	res0				: UINT; 
	stFromTime			: ST_BA_Time;
	stToTime			: ST_BA_Time;
	stRecipient			: ST_BACnet_Recipient;
	nProcessId			: UDINT;
	nEventTransitions	: ST_BACnet_EventTransitionBits;
	{attribute 'hide'}
	res1				: UINT; 
	bIssueConfirmed		: BOOL;
	{attribute 'hide'}
	res2				: ARRAY[0..2] OF BYTE;
END_STRUCT
END_TYPE

// DUTs/Types/Properties/Recipient/ST_BACnet_Recipient
{attribute 'hide'}
TYPE ST_BACnet_Recipient :
STRUCT
	eRecipientChoice: E_BACnet_RecipientChoice;
	{attribute 'hide'}
	res0 : UINT := 0;
	stEntry 		: ST_BACnet_RecipientEntry;
END_STRUCT
END_TYPE

// DUTs/Types/Properties/Recipient/ST_BACnet_RecipientEntry
{attribute 'hide'}
TYPE ST_BACnet_RecipientEntry :
UNION
	nDeviceInstance	: UDINT;
//	tDeviceId	: T_BACnet_ObjectIdentifier := 16#FFFFFFFF;
	stNetAddr	: ST_BACnet_Address;
END_UNION
END_TYPE

// DUTs/Types/Properties/Recipient/ST_BACnet_ValidDays
{attribute 'hide'}
TYPE ST_BACnet_ValidDays :
STRUCT
	{attribute 'hide'}
	res0			: BYTE;	
	{attribute 'hide'}
	res1			: BIT;
	
	bSunday			: BIT;
	bSaturday		: BIT;
	bFriday			: BIT;
	bThursday		: BIT;
	bWednesday		: BIT;
	bTuesday		: BIT;
	bMonday			: BIT;
END_STRUCT
END_TYPE

// DUTs/Types/Properties/References/ST_BACnet_ObjectPropertyReference
TYPE ST_BACnet_ObjectPropertyReference :
STRUCT
	iObject				: I_BACnet_Object;
	tObjectID			: T_BACnet_ObjectIdentifier		:= 16#FFFFFFFF;
	
	ePropertyId			: E_BACnetPropIdentifier		:= E_BACnetPropIdentifier.PropPresentValue;
END_STRUCT
END_TYPE

// DUTs/Types/Properties/Scheduler/ST_BACnet_EnumerationValueType
TYPE ST_BACnet_EnumerationValueType :
STRUCT
	choice 	   : E_BACnet_EnumerationValueChoice;
	enumValue  : UDINT;
END_STRUCT
END_TYPE

// DUTs/Types/Properties/Scheduler/ST_BACnet_SchedCalendar
TYPE ST_BACnet_SchedCalendar :
STRUCT
	iRefCalendar	: I_BACnet_Object;
	tRefCalendarID	: T_BACnet_ObjectIdentifier := 16#FFFFFFFF;
	
	{attribute 'hide'}
	nReserve		: DWORD; // May be used in future as a sequence-index
	
	eEventPriority	: E_BACnet_Priority := E_BACnet_Priority.eP1;
	stEntry			: ARRAY[1 .. BACnet_Param.nSched_EntryCount] OF ST_BA_SchedEntry;
END_STRUCT
END_TYPE

// DUTs/Types/Properties/Scheduler/ST_BACnet_SchedException
TYPE ST_BACnet_SchedException :
STRUCT
	eType			: E_BA_DateValChoice := E_BA_DateValChoice.Invalid;
	uDate			: U_BA_DateVal;
	
	{attribute 'hide'}
	nReserve		: DWORD;			// May be used in future as a sequence-index
	
	nEventPriority	: UDINT := 1;
	stEntry			: T_BACnet_SchedExceptionEntryList;
END_STRUCT
END_TYPE

// DUTs/Types/Properties/Scheduler/ST_BACnet_SpecialEvent
TYPE ST_BACnet_SpecialEvent :
STRUCT
	eEventChoice		: E_BACnet_SpecialEventChoice;
	{attribute 'hide'}
	_res1				: UINT;
	eCalEntryChoice		: E_BACnet_CalendarEntryChoice;
	{attribute 'hide'}
	_res2				: UINT;
	uCalEntry			: U_BA_DateVal;				// BACnetObjectIdentifier calendarReference;
	nEventPriority		: UDINT;
	{attribute 'hide'}
	_res3				: UDINT;
END_STRUCT
END_TYPE

// DUTs/Types/Properties/Scheduler/ST_BACnet_SpecialEventList
TYPE ST_BACnet_SpecialEventList :
STRUCT
	nEntrySize	: DWORD;
	nRes		: DWORD;
	stEvent 		: ST_BACnet_SpecialEvent;
END_STRUCT
END_TYPE

// DUTs/Types/Properties/Scheduler/T_BACnet_SchedCalendar
TYPE T_BACnet_SchedCalendar : ARRAY[1 .. BACnet_Param.nSched_CalendarCount] OF ST_BACnet_SchedCalendar; END_TYPE

// DUTs/Types/Properties/Scheduler/T_BACnet_SchedExceptionEntryList
TYPE T_BACnet_SchedExceptionEntryList : ARRAY[1 .. BACnet_Param.nSched_EntryCount] OF ST_BA_SchedEntry; END_TYPE

// DUTs/Types/Properties/Scheduler/T_BACnet_SchedExceptionList
TYPE T_BACnet_SchedExceptionList : ARRAY[1 .. BACnet_Param.nSched_ExceptionCount] OF ST_BACnet_SchedException; END_TYPE

// DUTs/Types/Properties/Scheduler/T_BACnet_SchedWeek
TYPE T_BACnet_SchedWeek : ARRAY[E_BA_Weekday.First .. E_BA_Weekday.Last, 1 .. BACnet_Param.nSched_EntryCount] OF ST_BA_SchedEntry; END_TYPE

// DUTs/Types/Properties/TLog/T_BACnet_TLogBuffer
TYPE T_BACnet_TLogBuffer : ARRAY [1 .. BACnet_Param.nTLog_ArraySize] OF ST_BA_TrendEntry; END_TYPE

// DUTs/Types/Properties/ST_BACnet_EventTransitionBits
{attribute 'hide'}
TYPE ST_BACnet_EventTransitionBits :
STRUCT
	{attribute 'hide'}
	_unusedBits : BYTE;
	{attribute 'hide'}
	res0 : BIT;
	{attribute 'hide'}
	res1 : BIT;
	{attribute 'hide'}
	res2 : BIT;
	{attribute 'hide'}
	res3 : BIT;
	{attribute 'hide'}
	res4 : BIT;
	bToNormal : BIT;
	bToFault : BIT;
	bToOffNormal : BIT;
END_STRUCT
END_TYPE

// DUTs/Types/Properties/ST_BACnet_ServicesSupportedBits
{attribute 'hide'}
TYPE ST_BACnet_ServicesSupportedBits :
STRUCT
	_unusedBits : BYTE;

	bSuppAtomicWriteFile  : BIT;
	bSuppAtomicReadFile  : BIT;
	bSuppSubscribeCOV  : BIT;
	bSuppGetEnrollmentSummary  : BIT;
	bSuppGetAlarmSummary  : BIT;
	bSuppConfirmedEventNotification  : BIT;
	bSuppConfirmedCOVNotification  : BIT;	
	bSuppAcknowledgeAlarm : BIT;

	bSuppWriteProperty : BIT;
	bSuppReadPropertyMultiple  : BIT;
	bSuppReadPropertyConditional  : BIT;
	bSuppReadProperty  : BIT;
	bSuppDeleteObject : BIT;
	bSuppCreateObject  : BIT;
	bSuppRemoveListElement  : BIT;
	bSuppAddListElement  : BIT;

	bSuppVtData  : BIT;
	bSuppVtClose : BIT;
	bSuppVtOpen  : BIT;
	bSuppReinitializeDevice  : BIT;	
	bSuppConfirmedTextMessage : BIT;
	bSuppConfirmedPrivateTransfer : BIT;
	bSuppDeviceCommunicationControl  : BIT;
	bSuppWritePropertyMultiple  : BIT;

	bSuppUnconfirmedTextMessage  : BIT;
	bSuppUnconfirmedPrivateTransfer  : BIT;
	bSuppUnconfirmedEventNotification  : BIT;	
	bSuppUnconfirmedCOVNotification  : BIT;
	bSuppIHave  : BIT;
	bSuppIAm  : BIT;
	bSuppRequestKey  : BIT;	
	bSuppAuthenticate  : BIT;

	bSuppGetEventInformation  : BIT;
	bSuppSubscribeCOVProperty  : BIT;
	bSuppLifeSafetyOperation  : BIT;
	bSuppUtcTimeSynchronization  : BIT;
	bSuppReadRange  : BIT;
	bSuppWhoIs  : BIT;
	bSuppWhoHas  : BIT;	
	bSuppTimeSynchronization  : BIT;
	
	_reserved : BYTE;
END_STRUCT
END_TYPE

// DUTs/Types/Properties/T_BACnet_ObjectIdentifier
TYPE T_BACnet_ObjectIdentifier : DWORD; END_TYPE

// DUTs/Types/Properties/T_BACnet_StateText
TYPE T_BACnet_StateText : STRING(BACnet_Param.nStateText_Length); END_TYPE

// DUTs/Types/Remote/[Internal]/ST_BACnetRM_CmdRealValue
TYPE INTERNAL ST_BACnetRM_CmdRealValue :
STRUCT
	fValue : REAL;
	bNull : BOOL;
END_STRUCT
END_TYPE

// DUTs/Types/Remote/[Internal]/ST_BACnetRM_FifoEntry
TYPE INTERNAL ST_BACnetRM_FifoEntry :
UNION
	fbRead : POINTER TO FB_BACnetRM_ReadProperty;
	fbWrite : POINTER TO FB_BACnetRM_WriteProperty;
END_UNION
END_TYPE

// DUTs/Types/Remote/[Internal]/ST_BACnetRM_LastWriteValue
TYPE INTERNAL ST_BACnetRM_LastWriteValue :
UNION
	stCmdValue : ST_BACnetRM_CmdRealValue;
	n8Value : BYTE;
	n16Value : UINT;
	n32Value : UDINT;
	nOther : POINTER TO BYTE;
END_UNION
END_TYPE

// DUTs/Types/Remote/[Internal]/ST_BACnetRM_PropertyValueList
{attribute 'enable_dynamic_creation'}
TYPE INTERNAL ST_BACnetRM_PropertyValueList :
STRUCT
	nEntrySize		: DWORD; (* 0x80000000 -> next entry *)
	{attribute 'hide'}
	nRes			: DWORD;
	nValidFields	: DWORD;
	ePropID			: E_BACnetPropIdentifier;		// [0]
	nArrayIndex		: DWORD;						// [1] (Optional)
	nPriority		: DWORD;						// [3] Unsigned (1 .. 16) (Optional -- used only when property is commandable)
	nValueSize		: DWORD;
	nDataType		: DWORD;
	
	// Data
END_STRUCT
END_TYPE

// DUTs/Types/Remote/[Internal]/ST_BACnetRM_ReadEntry
{attribute 'enable_dynamic_creation'}
TYPE INTERNAL ST_BACnetRM_ReadEntry :
STRUCT
	iObject 	: I_BACnetRM_BaseObject;
	ePropID 	: E_BACnetPropIdentifier;
	
	pData 		: PVOID;
	nData 		: UDINT;
	nIndex 		: UDINT := 16#FFFFFFFF;
	
	fbReadProp	: POINTER TO FB_BACnetRM_ReadProperty;
	
	_bError		: BOOL;										// Temporary error flag
END_STRUCT
END_TYPE

// DUTs/Types/Remote/[Internal]/ST_BACnetRM_ReqPtr
TYPE INTERNAL ST_BACnetRM_ReqPtr :
UNION
	nByte : POINTER TO BYTE;
	pPtr : PVOID;
	iReq : I_BACnetRM_Req;
	
	fbBase : POINTER TO FB_BACnetRM_ReqBasic;
	fbCov : POINTER TO FB_BACnetRM_ReqCov;
	fbRead : POINTER TO FB_BACnetRM_ReqRead;
	fbRpm : POINTER TO FB_BACnetRM_ReqRpm;
	fbWrite : POINTER TO FB_BACnetRM_ReqWrite;
	fbWpm : POINTER TO FB_BACnetRM_ReqWpm;
END_UNION
END_TYPE

// DUTs/Types/Remote/[Internal]/ST_BACnetRM_RpmListEntry
{attribute 'enable_dynamic_creation'}
TYPE INTERNAL ST_BACnetRM_RpmListEntry :
STRUCT
	nEntrySize 	: DWORD;					// 0x80000000 -> next entry
	tObjectID	: T_BACnet_ObjectIdentifier;
	ePropID		: E_BACnetPropIdentifier;
	nValidBits	: DWORD;
	nArrayIndex	: DWORD;
	nPriority	: DWORD;
END_STRUCT
END_TYPE

// DUTs/Types/Remote/[Internal]/ST_BACnetRM_ScanParameter
TYPE INTERNAL ST_BACnetRM_ScanParameter :
STRUCT
	bRescrictID	 : BIT;
	bRestrictNet : BIT;
	bLocalBroadcast : BIT;
	nNetNr : UINT;
	nStartID : UDINT;
	nEndID : UDINT;
END_STRUCT
END_TYPE

// DUTs/Types/Remote/[Internal]/ST_BACnetRM_WriteEntry
{attribute 'enable_dynamic_creation'}
TYPE INTERNAL ST_BACnetRM_WriteEntry :
STRUCT
	iObject 	: I_BACnetRM_BaseObject;
	ePropID 	: E_BACnetPropIdentifier;
	
	pData 		: PVOID;
	pEnable 	: POINTER TO BOOL;
	pNull 		: POINTER TO BOOL;
	nData 		: UDINT;
	fCOVIncrement : REAL := 0.0;
	nPriority 	: UDINT := 16;
END_STRUCT
END_TYPE

// DUTs/Types/Remote/ST_BACnetRM_ScanResult
TYPE ST_BACnetRM_ScanResult :
STRUCT
	tDeviceObjIdentifier : T_BACnet_ObjectIdentifier;
	nNetAddress : ARRAY [0..11] OF BYTE;
	nNetID : UINT;
	{attribute 'hide'}
	nRes : UINT;
	tIPAddr : IPADDR;	
	nUDPPort : UINT;		
	nVendorID : UINT;
	tMaxAddr : ETHERNET_ADDRESS;
END_STRUCT
END_TYPE

// TEST/TestPackage/TEMPLATES/HeatSupply/E_xEnergyLvl
{attribute 'qualified_only'}
TYPE E_xEnergyLvl :
(
	Protection		:= 1,
	Economy			:= 2,
	Comfort			:= 3
) UDINT;
END_TYPE

// TEST/TestPackage/TEMPLATES/HeatSupply/E_xEnergyLvlA
{attribute 'qualified_only'}
TYPE E_xEnergyLvlA :
(
	Automatic		:= 1,
	Protection		:= (E_xEnergyLvl.Protection + Automatic),
	Economy			:= (E_xEnergyLvl.Economy + Automatic),
	Comfort			:= (E_xEnergyLvl.Comfort + Automatic)
) UDINT;
END_TYPE

// GVLs/BACnet_Globals
{attribute 'qualified_only'}
VAR_GLOBAL
	{region 'Default Objects'}
		DefaultAdapter					: FB_BACnet_Adapter;									// Global linkable BACnet adapter
		DefaultServer					: FB_BACnet_Server;										// Global linkable BACnet device
	{endregion}
END_VAR
VAR_GLOBAL CONSTANT
	{region 'Commands'}
		sCmd_ConcatTitle				: STRING(5)							:= '\/';			// Command for inheriting path in entered title.
	{endregion}

	{region 'Placeholder'}
		{region 'Type Ranges'}
			nRange_ObjectTypeFirst		: INT								:= E_BACnetObjType.ObjAnalogInput;
			nRange_ObjectTypeLast		: INT								:= E_BACnetObjType.ObjChannel;
			nRange_ObjectTypeCount		: INT								:= (nRange_ObjectTypeLast - nRange_ObjectTypeFirst + 1);
		{endregion}
		{region 'Types'}
			nBACnetString_MaxLength		: INT								:= 256;
			nBACnetObjId_None			: T_BACnet_ObjectIdentifier			:= 16#FFFFFFFF;
		{endregion}
	{endregion}

	{region 'Object specification'}
		sSpec_ObjectTypeShortcut		: ARRAY [nRange_ObjectTypeFirst .. nRange_ObjectTypeLast] OF STRING(6) := [
											(* 	AnalogInput					*)	'AI',
											(* 	AnalogOutput				*)	'AO',
											(* 	AnalogValue					*)	'AV',
											(* 	BinaryInput					*)	'BI',
											(* 	BinaryOutput				*)	'BO',
											(* 	BinaryValue					*)	'BV',
											(* 	Calendar					*)	'CAL',
											(* 	Command						*)	'CMD',
											(* 	Device						*)	'DEV',
											(* 	EventEnrollment				*)	'EE',
											(* 	File						*)	'FILE',
											(* 	Group						*)	'GROUP',
											(* 	Loop						*)	'LOOP',
											(* 	MultiStateInput				*)	'MI',
											(* 	MultiStateOutput			*)	'MO',
											(* 	NotificationClass			*)	'NC',
											(* 	Program						*)	'PROG',
											(* 	Schedule					*)	'SCHED',
											(* 	Averaging					*)	'AVG',
											(* 	MultiStateValue				*)	'MV',
											(* 	TrendLog					*)	'TLOG',
											(* 	LifeSafetyPoint				*)	'LSP',
											(* 	LifeSafetyZone				*)	'LSZ',
											(* 	Accumulator					*)	'ACC',
											(* 	PulseConverter				*)	'PC',
											(* 	EventLog					*)	'ELOG',
											(* 	GlobalGroup					*)	'GGROUP',
											(* 	TrendLogMultiple			*)	'TLM',
											(* 	LoadControl					*)	'LOAD',
											(* 	StructuredView				*)	'VIEW',
											(* 	AccessDoor					*)	'DOOR',
											(* 	<Reserved>					*)	'',
											(* 	AccessCredential			*)	'AC',
											(* 	AccessPoint					*)	'AP',
											(* 	AccessRights				*)	'AR',
											(* 	AccessUser					*)	'AU',
											(* 	AccessZone					*)	'AZ',
											(* 	CredentialDataInput			*)	'CDI',
											(* 	NetworkSecurity				*)	'NS',
											(* 	BitStringValue				*)	'BIV',
											(* 	CharacterStringValue		*)	'CV',
											(* 	DatePatternValue			*)	'DPV',
											(* 	DateValue					*)	'DV',
											(* 	DateTimePatternValue		*)	'DTPV',
											(* 	DateTimeValue				*)	'DV',
											(* 	IntegerValue				*)	'IV',
											(* 	LargeAnalogValue			*)	'LAV',
											(* 	OctetStringValue			*)	'OV',
											(* 	PositiveIntegerValue		*)	'PIV',
											(* 	TimePatternValue			*)	'TPV',
											(* 	TimeValue					*)	'TV',
											(* 	NetworkPort					*)	'NP',
											(* 	AlertEnrollment				*)	'AE',
											(* 	Channel						*)	'C'
										];
	{endregion}
END_VAR
VAR_GLOBAL CONSTANT INTERNAL
	{region 'Placeholder'}
		{region 'AMS'}
			tInvalidAmsNetId			: T_AmsNetId						:= '0.0.0.0.0.0';
		{endregion}
		{region 'Types'}
			// (BETA) ... will be removed when ADS communication is removed
			{attribute 'hide'}
			nDataField_MaxDayEntry				: UINT						:= 19;
			{attribute 'hide'}
			nDataField_MaxExSchEntries			: UINT						:= 9;
			{attribute 'hide'}
			nDataField_MaxTimeValues			: UINT						:= 9;
			{attribute 'hide'}
			nDataField_MaxObjIdList				: UINT						:= 1999;
			{attribute 'hide'}
			nDataField_MaxLogBufferEntries		: UINT						:= 499;
			{attribute 'hide'}
			nDataField_MaxEventLogBufferEntries	: UINT						:= 500;
		{endregion}
	{endregion}
END_VAR

VAR_GLOBAL
	{region 'Internal'}
		{attribute 'hide'}
		stADSBuffer						: ST_BACnet_GlobalAdsBuffer;							// ADS read/write buffer for dynamic sized properties
		{attribute 'hide'}
		bDefaultBuffer					: ARRAY [0 .. BACnet_Param.nADS_BufferSize] OF BYTE;	// 8kByte common ADS buffer used by function blocks that access BACnet over ADS
	{endregion}
END_VAR

// GVLs/BACnet_Param
{attribute 'qualified_only'}
VAR_GLOBAL CONSTANT
	{region 'ADS'}
		tADS_TimeOut							: TIME					:= T#15S;
		nADS_BufferSize							: INT					:= 25535;								// Default 24 kByte buffer
	{endregion}
	{region 'Priorities'}
		nPrio_LifeSafety 						: BYTE					:= 1;
		nPrio_Critical							: BYTE					:= 5;
		nPrio_ManLocal							: BYTE					:= 7;
		nPrio_ManRemote 						: BYTE					:= 8;
		nPrio_Program 	 						: BYTE					:= 15;
		nPrio_Default	 	 					: BYTE					:= 17;									// No priority used

		nRemotePrio_Default						: BYTE					:= 8;									// Default priority for priority enabled remote-objects
	{endregion}
		
	{region 'Event-Management'}
		sEvtMgmt_AckMsgRemote					: STRING				:= 'Acknowledged by remote user.';		// Text to indicate acknowledgement via remote access.
		sEvtMgmt_AckMsgPLC						: STRING				:= 'Acknowledged by PLC.';				// Text to indicate acknowledgement via PLC logic.
	{endregion}
	{region 'Titles'}
		sSeparator_ObjectName					: STRING				:= '_';									// Separator to be used when building Inherited object names
		sSeparator_Description					: STRING				:= ' - ';								// Separator to be used when building Inherited descriptions
		sSeparator_EventMessageText				: STRING				:= ' - ';								// Separator to be used when building Inherited event message texts
	{endregion}
		 
	{region 'Objects'}
		{region 'General'}
			nStateText_Length					: UDINT					:= 40;									// Max. count of string characters in state texts (e.g. Multustate-StateText, Binary-In/ActiveText)
			bStateText_WriteProtect				: BOOL					:= FALSE;
		{endregion}
		{region 'Multistate'}
			nMultistate_StateCount				: UDINT					:= 24;									// Count of state entries
		{endregion}
		{region 'EventLog'}
			nEventLog_ArraySize					: UDINT					:= 500;
		{endregion}
		{region 'TrendLog'}
			nTLog_ArraySize						: UDINT					:= 500;
		{endregion}
		{region 'Calendar'}
			nCal_DateListCount					: INT					:= 24;									// Count of date list entries ('T_BACnet_CalendarDateList')
		{endregion}
		{region 'NC'}
			nNC_RecipientArraySize				: INT					:= 19;									// Count of recipient entries
		{endregion}
		{region 'Scheduler'}
			nSched_PrioForWriting				: UDINT					:= 16;
						  
			nSched_EntryCount					: INT					:= 6;									// Count of entries in a weekday ('ST_BACnet_SchedWeekday') or an exception ('ST_BACnet_SchedException')
			nSched_CalendarCount				: INT					:= 3;									// Count of calendar references ('T_BACnet_SchedCalendar')
			nSched_ExceptionCount				: INT					:= 24;									// Count of exceptions ('T_BACnet_SchedException')

			eSched_BType						: E_BACnet_SchedBType	:= E_BACnet_SchedBType.eBool;			// Internal datatype of boolean schedulers
		{endregion}
	{endregion}
END_VAR

// TEST/TestPackage/TEMPLATES/Const
{attribute 'qualified_only'}
VAR_GLOBAL CONSTANT
	rClsZero        : REAL := 0.00001;//Comparison value to prevent a division by zero
						
	nNoActvPrio	: UDINT	:= 4294967295;//Value of the constant indicates that no priority is active	
	
	nTiSec        : UDINT := 4294966;
	nTiMin        : UDINT := 71582;

	wSUNDAY         : WORD := 0;//Constant value for Sunday
	wMONDAY         : WORD := 1;//Constant value for Monday
	wTUESDAY        : WORD := 2;//Constant value for Tuesday
	wWEDNESDAY      : WORD := 3;//Constant value for Wednesday
	wTHURSDAY       : WORD := 4;//Constant value for Thursday
	wFRIDAY         : WORD := 5;//Constant value for Friday
	wSATURDAY       : WORD := 6;//Constant value for Saturday

	TimeValue24h_ms : UDINT := 86400000;//Time value for 24 hours in ms
END_VAR

// Version/Global_Version
{attribute 'TcGenerated'}
{attribute 'no-analysis'}
{attribute 'linkalways'}
// This function has been automatically generated from the project information.
VAR_GLOBAL CONSTANT
	{attribute 'const_non_replaced'}
	stLibVersion_Tc3_BACnetRev14 : ST_LibVersion := (iMajor := 4, iMinor := 0, iBuild := 11, iRevision := 0, nFlags := 0, sVersion := '4.0.11.0');
END_VAR

// DUTs/Interfaces/Remote/[Base]/I_BACnetRM_Object
INTERFACE I_BACnetRM_Object EXTENDS I_BACnetRM_BaseObject

END_INTERFACE

// DUTs/Interfaces/Remote/[Internal]/I_BACnetRM_BaseObject
INTERFACE I_BACnetRM_BaseObject

{attribute 'hide'}
METHOD OnCOV
VAR_INPUT
	ePropID		: E_BACnetPropIdentifier;
END_VAR
END_METHOD

{attribute 'hide'}
METHOD OnReqError
VAR_INPUT
	iRequest		: I_BACnetRM_Req;
	
	eResult			: E_BACnetRM_Error;
	sLogCode		: STRING			:= '';
END_VAR
END_METHOD

PROPERTY Error : BOOL
GET
END_GET
END_PROPERTY

PROPERTY ObjectID : T_BACnet_ObjectIdentifier
GET
END_GET
END_PROPERTY

PROPERTY ObjectInstance : UDINT
GET
END_GET
END_PROPERTY

PROPERTY ObjectType : E_BACnetObjType
GET
END_GET
END_PROPERTY

PROPERTY Ready : BOOL
GET
END_GET
END_PROPERTY

END_INTERFACE

// DUTs/Interfaces/Remote/I_BACnetRM_Req
{attribute 'c++_compatible'}
INTERFACE I_BACnetRM_Req

{attribute 'hide'}
METHOD Send : BOOL
VAR_INPUT
END_VAR
END_METHOD

METHOD GetRequestType : E_BACnetRM_RequestType
VAR_INPUT
END_VAR
END_METHOD

METHOD IsReady : BOOL
VAR_INPUT
END_VAR
END_METHOD

END_INTERFACE

// DUTs/Interfaces/Remote/[Internal]/I_BACnetRM_ObjectOwner
{attribute 'hide'}
INTERFACE I_BACnetRM_ObjectOwner EXTENDS __SYSTEM.IQueryInterface

{attribute 'hide'}
METHOD OnBACnetRMObjectCOV
VAR_INPUT
	ePropID		: E_BACnetPropIdentifier;
END_VAR
END_METHOD

{attribute 'hide'}
METHOD OnBACnetRMObjectStateChanged
END_METHOD

{attribute 'suppress_wrn_C0410'}
{attribute 'hide'}
PROPERTY LogMsg : REFERENCE TO FB_BA_LogMessage
GET
END_GET
END_PROPERTY

END_INTERFACE

// DUTs/Interfaces/Server/[Base]/I_BACnet_Object
INTERFACE I_BACnet_Object EXTENDS I_BACnet_BaseObject

PROPERTY Parent : I_BACnet_View
GET
END_GET
SET
END_SET
END_PROPERTY

PROPERTY Description : T_MaxString
GET
END_GET
SET
END_SET
END_PROPERTY

PROPERTY ObjectName : T_MaxString
GET
END_GET
SET
END_SET
END_PROPERTY

END_INTERFACE

// DUTs/Interfaces/Server/[Internal]/I_BACnet_BaseObject
{attribute 'hide'}
INTERFACE I_BACnet_BaseObject EXTENDS I_BA_SupplementObject

PROPERTY Error : BOOL
GET
END_GET
END_PROPERTY

PROPERTY ObjectID : T_BACnet_ObjectIdentifier
GET
END_GET
END_PROPERTY

PROPERTY ObjectInstance : UDINT
GET
END_GET
END_PROPERTY

PROPERTY ObjectType : E_BACnetObjType
GET
END_GET
END_PROPERTY

PROPERTY Ready : BOOL
GET
END_GET
END_PROPERTY

METHOD ReadProperty : HRESULT
VAR_INPUT
	ePropID : E_BACnetPropIdentifier;
	pData : PVOID;
	nData : POINTER TO DINT;
END_VAR
END_METHOD

METHOD SyncPropertyCOV : BOOL
VAR_IN_OUT
	bChangeTrig : BOOL;
END_VAR
VAR_INPUT
	ePropertyID : E_BACnetPropIdentifier;
END_VAR
END_METHOD

METHOD WriteProperty : HRESULT
VAR_INPUT
	ePropID : E_BACnetPropIdentifier;
	pData : PVOID;
	nData : DINT;
END_VAR
END_METHOD

END_INTERFACE

// DUTs/Interfaces/Server/Misc/I_BACnet_View
INTERFACE I_BACnet_View EXTENDS I_BACnet_Object

END_INTERFACE

// DUTs/Interfaces/Server/[Internal]/I_BACnet_ObjectOwner
{attribute 'hide'}
INTERFACE I_BACnet_ObjectOwner EXTENDS __SYSTEM.IQueryInterface

{attribute 'hide'}
METHOD OnBACnetObjectStateChanged
VAR_INPUT
	tState			: TCOM_STATE;
END_VAR
END_METHOD

{attribute 'suppress_wrn_C0410'}
{attribute 'hide'}
PROPERTY LogMsg : REFERENCE TO FB_BA_LogMessage
GET
END_GET
END_PROPERTY

{attribute 'hide'}
PROPERTY SymbolPath : REFERENCE TO T_MaxString
GET
END_GET
END_PROPERTY

END_INTERFACE

// DUTs/Interfaces/Server/Misc/I_BACnet_Cal
INTERFACE I_BACnet_Cal EXTENDS I_BACnet_Object

END_INTERFACE

// POUs/Helper/[internal]/Calendar/F_BACnet_CopyDateListEntry
{attribute 'hide'} // [Workaround] Not hidden when lib is included
FUNCTION INTERNAL F_BACnet_ToDateListEntry : BOOL
VAR_INPUT
	stEntry		: POINTER TO ST_BA_CalendarEntry;
END_VAR
VAR_OUTPUT
	stResult	: ST_BACnet_CalendarEntry;
END_VAR

IF (stEntry <> 0) AND_THEN (F_BA_IsDateValChoiceValid(stEntry^.eType)) THEN
	// Clear contents:
	MEMSET(ADR(stResult), 0, SIZEOF(ST_BACnet_CalendarEntry));
 
	CASE (stEntry^.eType) OF
		E_BA_DateValChoice.eDate:
			stResult.uCalEntry.stDate := stEntry^.uDate.stDate;
		E_BA_DateValChoice.eDateRange:
			stResult.uCalEntry.stDateRange := stEntry^.uDate.stDateRange;
		E_BA_DateValChoice.eWeekNDay:
			stResult.uCalEntry.stWeekNDay := stEntry^.uDate.stWeekNDay;
	ELSE
		RETURN;
	END_CASE
	
	stResult.eEventChoice := (stEntry^.eType-1);
	
	F_BACnet_ToDateListEntry := TRUE;
END_IF

END_FUNCTION

// POUs/Helper/[internal]/Remote/F_BACnetRM_IsErrorSet
{attribute 'hide'}
FUNCTION F_BACnetRM_IsErrorSet : BOOL
VAR_INPUT
	stResult	: POINTER TO SendDataRequestResult;
END_VAR
VAR
END_VAR

